  MoveL 3948 to (-81.04, 7.67, -135.54) mm, rotated rx 42.04 ry 15.1 rz -114.75 deg; joints [-14.521, -47.036, 111.718, 147.61, 50.435, -29.895, -355]
  MoveL 3949 to (-78.95, 8.33, -135.66) mm, rotated rx 42.04 ry 15.1 rz -114.75 deg; joints [-14.521, -46.888, 111.628, 147.636, 50.484, -29.936, -355]
  MoveL 3950 to (-78.47, 8.53, -135.68) mm, rotated rx 42.04 ry 15.1 rz -114.75 deg; joints [-14.52, -46.852, 111.603, 147.642, 50.493, -29.944, -355]
  MoveL 3951 to (-78.06, 8.74, -135.73) mm, rotated rx 42.04 ry 15.1 rz -114.75 deg; joints [-14.52, -46.82, 111.578, 147.645, 50.499, -29.949, -355]
  MoveL 3952 to (-77.68, 8.96, -135.8) mm, rotated rx 42.04 ry 15.1 rz -114.75 deg; joints [-14.521, -46.79, 111.553, 147.645, 50.503, -29.951, -355]
  MoveL 3953 to (-77.28, 9.16, -135.86) mm, rotated rx 42.04 ry 15.1 rz -114.75 deg; joints [-14.522, -46.759, 111.528, 147.647, 50.509, -29.956, -355]
  MoveL 3954 to (-76.86, 9.36, -135.89) mm, rotated rx 42.04 ry 15.1 rz -114.75 deg; joints [-14.522, -46.727, 111.504, 147.651, 50.515, -29.961, -355]
  MoveL 3955 to (-72.52, 11.13, -135.9) mm, rotated rx 42.04 ry 15.1 rz -114.75 deg; joints [-14.508, -46.408, 111.285, 147.712, 50.597, -30.037, -355]
  MoveL 3956 to (-72.12, 11.31, -135.92) mm, rotated rx 42.04 ry 15.1 rz -114.75 deg; joints [-14.507, -46.377, 111.263, 147.716, 50.603, -30.043, -355]
  MoveL 3957 to (-71.68, 11.49, -135.93) mm, rotated rx 42.04 ry 15.1 rz -114.75 deg; joints [-14.506, -46.345, 111.24, 147.722, 50.611, -30.05, -355]
  MoveL 3958 to (-70.72, 11.88, -135.93) mm, rotated rx 42.04 ry 15.1 rz -114.75 deg; joints [-14.503, -46.274, 111.191, 147.735, 50.629, -30.066, -355]
  MoveL 3959 to (-70.2, 12.11, -135.94) mm, rotated rx 42.04 ry 15.1 rz -114.75 deg; joints [-14.502, -46.235, 111.163, 147.742, 50.638, -30.075, -355]
  MoveL 3960 to (-69.65, 12.36, -135.96) mm, rotated rx 42.04 ry 15.1 rz -114.75 deg; joints [-14.5, -46.194, 111.132, 147.748, 50.646, -30.082, -355]
  MoveL 3961 to (-69.07, 12.68, -135.99) mm, rotated rx 42.04 ry 15.1 rz -114.75 deg; joints [-14.499, -46.148, 111.095, 147.753, 50.653, -30.089, -355]
  MoveL 3962 to (-68.53, 13.06, -136.01) mm, rotated rx 42.04 ry 15.1 rz -114.75 deg; joints [-14.497, -46.103, 111.053, 147.757, 50.656, -30.092, -355]
  MoveL 3963 to (-68.02, 13.48, -136.03) mm, rotated rx 42.04 ry 15.1 rz -114.75 deg; joints [-14.494, -46.059, 111.009, 147.76, 50.655, -30.093, -355]
  MoveL 3964 to (-69.19, 12.88, -137.01) mm, rotated rx 42.04 ry 15.1 rz -114.75 deg; joints [-14.538, -46.143, 111.064, 147.695, 50.641, -30.053, -355]
  MoveL 3965 to (-68.73, 14.14, -137.43) mm, rotated rx 42.04 ry 15.1 rz -114.75 deg; joints [-14.546, -46.072, 110.943, 147.663, 50.6, -30.014, -355]
  MoveL 3966 to (-68.09, 15.49, -137.75) mm, rotated rx 42.04 ry 15.1 rz -114.75 deg; joints [-14.549, -45.989, 110.812, 147.639, 50.561, -29.981, -355]
  MoveL 3967 to (-67.25, 16.96, -137.99) mm, rotated rx 42.04 ry 15.1 rz -114.75 deg; joints [-14.548, -45.89, 110.669, 147.621, 50.523, -29.95, -355]
  MoveL 3968 to (-66.1, 18.76, -138.21) mm, rotated rx 42.04 ry 15.1 rz -114.75 deg; joints [-14.543, -45.761, 110.493, 147.605, 50.481, -29.919, -355]
  MoveL 3969 to (-64.92, 20.54, -138.32) mm, rotated rx 42.04 ry 15.1 rz -114.75 deg; joints [-14.535, -45.633, 110.319, 147.595, 50.441, -29.892, -355]
  MoveL 3970 to (-63.74, 22.32, -138.43) mm, rotated rx 42.04 ry 15.1 rz -114.75 deg; joints [-14.526, -45.504, 110.145, 147.585, 50.401, -29.864, -355]
  MoveL 3971 to (-62.57, 24.1, -138.66) mm, rotated rx 42.04 ry 15.1 rz -114.75 deg; joints [-14.522, -45.375, 109.968, 147.569, 50.36, -29.833, -355]
  MoveL 3972 to (-61.39, 25.88, -138.78) mm, rotated rx 42.04 ry 15.1 rz -114.75 deg; joints [-14.514, -45.247, 109.794, 147.558, 50.319, -29.805, -355]
  MoveL 3973 to (-60.21, 27.66, -139.01) mm, rotated rx 42.04 ry 15.1 rz -114.75 deg; joints [-14.51, -45.117, 109.617, 147.542, 50.278, -29.773, -355]
  MoveL 3974 to (-59.02, 29.43, -139.12) mm, rotated rx 42.04 ry 15.1 rz -114.75 deg; joints [-14.502, -44.988, 109.442, 147.531, 50.238, -29.745, -355]
  MoveL 3975 to (-57.83, 31.2, -139.24) mm, rotated rx 42.04 ry 15.1 rz -114.75 deg; joints [-14.494, -44.859, 109.267, 147.52, 50.197, -29.717, -355]
  MoveL 3976 to (-56.64, 32.97, -139.48) mm, rotated rx 42.04 ry 15.1 rz -114.75 deg; joints [-14.491, -44.729, 109.09, 147.503, 50.156, -29.686, -355]
  MoveL 3977 to (-55.48, 34.65, -139.58) mm, rotated rx 42.04 ry 15.1 rz -114.75 deg; joints [-14.483, -44.606, 108.923, 147.493, 50.118, -29.659, -355]
  MoveL 3978 to (-54.36, 36.29, -139.79) mm, rotated rx 42.04 ry 15.1 rz -114.75 deg; joints [-14.479, -44.484, 108.758, 147.478, 50.081, -29.63, -355]
  MoveL 3979 to (-53.04, 38.26, -139.95) mm, rotated rx 42.04 ry 15.1 rz -114.75 deg; joints [-14.471, -44.341, 108.562, 147.464, 50.034, -29.597, -355]
  MoveL 3980 to (-51.48, 40.49, -140.04) mm, rotated rx 42.04 ry 15.1 rz -114.75 deg; joints [-14.459, -44.175, 108.339, 147.453, 49.983, -29.563, -355]
  MoveL 3981 to (-50.32, 42.21, -140.1) mm, rotated rx 42.04 ry 15.1 rz -114.75 deg; joints [-14.449, -44.05, 108.168, 147.444, 49.942, -29.535, -355]
  MoveL 3982 to (-49.24, 43.8, -140.23) mm, rotated rx 42.04 ry 15.1 rz -114.75 deg; joints [-14.443, -43.933, 108.008, 147.432, 49.904, -29.508, -355]
  MoveL 3983 to (-48.12, 45.44, -140.34) mm, rotated rx 42.04 ry 15.1 rz -114.75 deg; joints [-14.435, -43.813, 107.844, 147.421, 49.866, -29.481, -355]
  MoveL 3984 to (-47.01, 47.05, -140.45) mm, rotated rx 42.04 ry 15.1 rz -114.75 deg; joints [-14.428, -43.694, 107.682, 147.41, 49.827, -29.453, -355]
  MoveL 3985 to (-45.85, 48.75, -140.52) mm, rotated rx 42.04 ry 15.1 rz -114.75 deg; joints [-14.419, -43.57, 107.511, 147.4, 49.787, -29.426, -355]
  MoveL 3986 to (-44.59, 50.58, -140.62) mm, rotated rx 42.04 ry 15.1 rz -114.75 deg; joints [-14.41, -43.435, 107.327, 147.389, 49.743, -29.395, -355]
  MoveL 3987 to (-43.19, 52.55, -140.88) mm, rotated rx 42.04 ry 15.1 rz -114.75 deg; joints [-14.406, -43.286, 107.125, 147.369, 49.697, -29.359, -355]
  MoveL 3988 to (-42.36, 54.62, -141.86) mm, rotated rx 42.04 ry 15.1 rz -114.75 deg; joints [-14.43, -43.163, 106.913, 147.299, 49.627, -29.284, -355]
  MoveL 3989 to (-42.38, 53.48, -142.35) mm, rotated rx 42.04 ry 15.1 rz -114.75 deg; joints [-14.457, -43.198, 107.005, 147.294, 49.682, -29.312, -355]
  MoveL 3990 to (-42.39, 52.89, -142.66) mm, rotated rx 42.04 ry 15.1 rz -114.75 deg; joints [-14.473, -43.216, 107.053, 147.288, 49.711, -29.326, -355]
  MoveL 3991 to (-42.38, 52.79, -142.81) mm, rotated rx 42.04 ry 15.1 rz -114.75 deg; joints [-14.479, -43.218, 107.059, 147.282, 49.716, -29.325, -355]
  MoveL 3992 to (-42.37, 53.13, -142.85) mm, rotated rx 42.04 ry 15.1 rz -114.75 deg; joints [-14.478, -43.206, 107.028, 147.274, 49.7, -29.312, -355]
  MoveL 3993 to (-42.37, 53.6, -142.86) mm, rotated rx 42.04 ry 15.1 rz -114.75 deg; joints [-14.476, -43.19, 106.987, 147.266, 49.678, -29.296, -355]
  MoveL 3994 to (-42.34, 54.08, -142.9) mm, rotated rx 42.04 ry 15.1 rz -114.75 deg; joints [-14.474, -43.173, 106.944, 147.256, 49.656, -29.278, -355]
  MoveL 3995 to (-42.31, 54.53, -142.96) mm, rotated rx 42.04 ry 15.1 rz -114.75 deg; joints [-14.473, -43.156, 106.903, 147.246, 49.635, -29.262, -355]
  MoveL 3996 to (-42.28, 54.99, -143) mm, rotated rx 42.04 ry 15.1 rz -114.75 deg; joints [-14.471, -43.139, 106.861, 147.237, 49.614, -29.245, -355]
  MoveL 3997 to (-42.26, 55.48, -143.02) mm, rotated rx 42.04 ry 15.1 rz -114.75 deg; joints [-14.469, -43.122, 106.818, 147.228, 49.591, -29.227, -355]
  MoveL 3998 to (-42.25, 58.1, -143.02) mm, rotated rx 42.04 ry 15.1 rz -114.75 deg; joints [-14.451, -43.036, 106.587, 147.182, 49.466, -29.133, -355]
  MoveL 3999 to (-42.24, 58.56, -143.04) mm, rotated rx 42.04 ry 15.1 rz -114.75 deg; joints [-14.449, -43.02, 106.546, 147.174, 49.445, -29.117, -355]
  MoveL 4000 to (-42.21, 58.94, -143.07) mm, rotated rx 42.04 ry 15.1 rz -114.75 deg; joints [-14.448, -43.005, 106.511, 147.166, 49.427, -29.103, -355]
  MoveL 4001 to (-42.19, 59.4, -143.09) mm, rotated rx 42.04 ry 15.1 rz -114.75 deg; joints [-14.445, -42.989, 106.47, 147.157, 49.405, -29.086, -355]
  MoveL 4002 to (-42.18, 60, -143.11) mm, rotated rx 42.04 ry 15.1 rz -114.75 deg; joints [-14.442, -42.968, 106.417, 147.146, 49.377, -29.064, -355]
  MoveL 4003 to (-42.13, 60.72, -143.17) mm, rotated rx 42.04 ry 15.1 rz -114.75 deg; joints [-14.439, -42.942, 106.352, 147.131, 49.344, -29.038, -355]
  MoveL 4004 to (-42.11, 61.34, -143.2) mm, rotated rx 42.04 ry 15.1 rz -114.75 deg; joints [-14.436, -42.92, 106.296, 147.119, 49.315, -29.016, -355]
  MoveL 4005 to (-42.11, 61.87, -143.2) mm, rotated rx 42.04 ry 15.1 rz -114.75 deg; joints [-14.433, -42.902, 106.249, 147.11, 49.29, -28.996, -355]
  MoveL 4006 to (-42.1, 63.44, -143.2) mm, rotated rx 42.04 ry 15.1 rz -114.75 deg; joints [-14.422, -42.849, 106.11, 147.082, 49.215, -28.939, -355]
  MoveL 4007 to (-41.79, 66.34, -143.54) mm, rotated rx 42.04 ry 15.1 rz -114.75 deg; joints [-14.416, -42.733, 105.843, 147.019, 49.086, -28.834, -355]
  MoveL 4008 to (-41.42, 67.58, -143.97) mm, rotated rx 42.04 ry 15.1 rz -114.75 deg; joints [-14.424, -42.667, 105.719, 146.982, 49.04, -28.788, -355]
  MoveL 4009 to (-40.9, 68.68, -144.57) mm, rotated rx 42.04 ry 15.1 rz -114.75 deg; joints [-14.439, -42.596, 105.603, 146.941, 49.006, -28.748, -355]
  MoveL 4010 to (-39.42, 70.47, -146.28) mm, rotated rx 42.04 ry 15.1 rz -114.75 deg; joints [-14.492, -42.439, 105.39, 146.851, 48.972, -28.681, -355]
  MoveL 4011 to (-37.35, 71.7, -148.68) mm, rotated rx 42.04 ry 15.1 rz -114.75 deg; joints [-14.574, -42.261, 105.204, 146.746, 48.986, -28.633, -355]
  MoveL 4012 to (-35.34, 72.15, -151.07) mm, rotated rx 42.04 ry 15.1 rz -114.75 deg; joints [-14.661, -42.113, 105.088, 146.655, 49.035, -28.613, -355]
  MoveL 4013 to (-34.6, 71.99, -152.01) mm, rotated rx 42.04 ry 15.1 rz -114.75 deg; joints [-14.698, -42.068, 105.073, 146.625, 49.069, -28.617, -355]
  MoveL 4014 to (-34.02, 71.57, -152.78) mm, rotated rx 42.04 ry 15.1 rz -114.75 deg; joints [-14.73, -42.044, 105.087, 146.604, 49.109, -28.629, -355]
  MoveL 4015 to (-33.8, 71.26, -153.1) mm, rotated rx 42.04 ry 15.1 rz -114.75 deg; joints [-14.744, -42.039, 105.105, 146.598, 49.132, -28.638, -355]
  MoveL 4016 to (-33.63, 70.89, -153.38) mm, rotated rx 42.04 ry 15.1 rz -114.75 deg; joints [-14.757, -42.039, 105.13, 146.594, 49.156, -28.65, -355]
  MoveL 4017 to (-33.4, 69.96, -153.81) mm, rotated rx 42.04 ry 15.1 rz -114.75 deg; joints [-14.78, -42.054, 105.202, 146.593, 49.209, -28.68, -355]
  MoveL 4018 to (-33.35, 68.77, -154.07) mm, rotated rx 42.04 ry 15.1 rz -114.75 deg; joints [-14.798, -42.088, 105.302, 146.603, 49.268, -28.719, -355]
  MoveL 4019 to (-33.47, 67.32, -154.15) mm, rotated rx 42.04 ry 15.1 rz -114.75 deg; joints [-14.811, -42.143, 105.431, 146.622, 49.334, -28.767, -355]
  MoveL 4020 to (-33.54, 66.8, -154.15) mm, rotated rx 42.04 ry 15.1 rz -114.75 deg; joints [-14.815, -42.164, 105.479, 146.63, 49.357, -28.784, -355]
  MoveL 4021 to (-33.64, 66.37, -154.1) mm, rotated rx 42.04 ry 15.1 rz -114.75 deg; joints [-14.816, -42.184, 105.519, 146.639, 49.374, -28.798, -355]
  MoveL 4022 to (-33.74, 65.95, -154.04) mm, rotated rx 42.04 ry 15.1 rz -114.75 deg; joints [-14.816, -42.204, 105.56, 146.647, 49.391, -28.813, -355]
  MoveL 4023 to (-33.82, 65.49, -154) mm, rotated rx 42.04 ry 15.1 rz -114.75 deg; joints [-14.818, -42.225, 105.603, 146.656, 49.41, -28.828, -355]
  MoveL 4024 to (-33.9, 65, -153.98) mm, rotated rx 42.04 ry 15.1 rz -114.75 deg; joints [-14.821, -42.246, 105.648, 146.664, 49.431, -28.844, -355]
  MoveL 4025 to (-33.98, 64.47, -153.98) mm, rotated rx 42.04 ry 15.1 rz -114.75 deg; joints [-14.824, -42.267, 105.697, 146.672, 49.454, -28.862, -355]
  MoveL 4026 to (-34.05, 63.95, -153.98) mm, rotated rx 42.04 ry 15.1 rz -114.75 deg; joints [-14.828, -42.288, 105.744, 146.68, 49.477, -28.879, -355]
  MoveL 4027 to (-34.1, 63.44, -153.99) mm, rotated rx 42.04 ry 15.1 rz -114.75 deg; joints [-14.832, -42.308, 105.789, 146.687, 49.5, -28.895, -355]
  MoveL 4028 to (-34.16, 62.95, -154) mm, rotated rx 42.04 ry 15.1 rz -114.75 deg; joints [-14.836, -42.327, 105.834, 146.694, 49.522, -28.912, -355]
  MoveL 4029 to (-34.23, 62.49, -153.98) mm, rotated rx 42.04 ry 15.1 rz -114.75 deg; joints [-14.838, -42.347, 105.876, 146.702, 49.541, -28.927, -355]
  MoveL 4030 to (-34.31, 62.04, -153.94) mm, rotated rx 42.04 ry 15.1 rz -114.75 deg; joints [-14.84, -42.367, 105.918, 146.71, 49.56, -28.942, -355]
  MoveL 4031 to (-34.42, 61.5, -153.89) mm, rotated rx 42.04 ry 15.1 rz -114.75 deg; joints [-14.842, -42.391, 105.968, 146.72, 49.582, -28.96, -355]
  MoveL 4032 to (-34.55, 60.81, -153.84) mm, rotated rx 42.04 ry 15.1 rz -114.75 deg; joints [-14.845, -42.422, 106.033, 146.732, 49.611, -28.983, -355]
  MoveL 4033 to (-34.66, 60.18, -153.81) mm, rotated rx 42.04 ry 15.1 rz -114.75 deg; joints [-14.848, -42.449, 106.091, 146.743, 49.638, -29.003, -355]
  MoveL 4034 to (-35.01, 57.58, -153.81) mm, rotated rx 42.04 ry 15.1 rz -114.75 deg; joints [-14.867, -42.554, 106.326, 146.781, 49.751, -29.088, -355]
  MoveL 4035 to (-35.11, 56.96, -153.78) mm, rotated rx 42.04 ry 15.1 rz -114.75 deg; joints [-14.869, -42.58, 106.383, 146.792, 49.777, -29.109, -355]
  MoveL 4036 to (-35.21, 56.41, -153.72) mm, rotated rx 42.04 ry 15.1 rz -114.75 deg; joints [-14.871, -42.604, 106.434, 146.802, 49.801, -29.127, -355]
  MoveL 4037 to (-35.25, 56.21, -153.57) mm, rotated rx 42.04 ry 15.1 rz -114.75 deg; joints [-14.867, -42.615, 106.455, 146.812, 49.809, -29.137, -355]
  MoveL 4038 to (-35.23, 56.33, -153.31) mm, rotated rx 42.04 ry 15.1 rz -114.75 deg; joints [-14.856, -42.611, 106.448, 146.824, 49.803, -29.14, -355]
  MoveL 4039 to (-35.13, 56.78, -152.9) mm, rotated rx 42.04 ry 15.1 rz -114.75 deg; joints [-14.837, -42.594, 106.414, 146.839, 49.784, -29.137, -355]
  MoveL 4040 to (-36.15, 56.59, -152.1) mm, rotated rx 42.04 ry 15.1 rz -114.75 deg; joints [-14.808, -42.665, 106.463, 146.863, 49.759, -29.135, -355]
  MoveL 4041 to (-37.5, 55.14, -151.88) mm, rotated rx 42.04 ry 15.1 rz -114.75 deg; joints [-14.81, -42.794, 106.619, 146.873, 49.782, -29.153, -355]
  MoveL 4042 to (-38.85, 53.66, -151.72) mm, rotated rx 42.04 ry 15.1 rz -114.75 deg; joints [-14.815, -42.923, 106.776, 146.881, 49.807, -29.171, -355]
  MoveL 4043 to (-40.23, 52.13, -151.57) mm, rotated rx 42.04 ry 15.1 rz -114.75 deg; joints [-14.821, -43.055, 106.938, 146.888, 49.833, -29.19, -355]
  MoveL 4044 to (-41.5, 50.75, -151.28) mm, rotated rx 42.04 ry 15.1 rz -114.75 deg; joints [-14.82, -43.177, 107.087, 146.902, 49.856, -29.21, -355]
  MoveL 4045 to (-42.91, 49.19, -151.09) mm, rotated rx 42.04 ry 15.1 rz -114.75 deg; joints [-14.824, -43.313, 107.253, 146.91, 49.882, -29.229, -355]
  MoveL 4046 to (-44.4, 47.54, -150.9) mm, rotated rx 42.04 ry 15.1 rz -114.75 deg; joints [-14.829, -43.456, 107.427, 146.918, 49.909, -29.249, -355]
  MoveL 4047 to (-45.9, 45.87, -150.82) mm, rotated rx 42.04 ry 15.1 rz -114.75 deg; joints [-14.838, -43.599, 107.601, 146.922, 49.937, -29.266, -355]
  MoveL 4048 to (-47.71, 43.83, -150.73) mm, rotated rx 42.04 ry 15.1 rz -114.75 deg; joints [-14.85, -43.774, 107.813, 146.925, 49.971, -29.288, -355]
  MoveL 4049 to (-49.01, 42.36, -150.62) mm, rotated rx 42.04 ry 15.1 rz -114.75 deg; joints [-14.857, -43.899, 107.966, 146.929, 49.996, -29.304, -355]
  MoveL 4050 to (-50.22, 41, -150.41) mm, rotated rx 42.04 ry 15.1 rz -114.75 deg; joints [-14.859, -44.017, 108.11, 146.939, 50.018, -29.322, -355]
  MoveL 4051 to (-51.55, 39.48, -150.22) mm, rotated rx 42.04 ry 15.1 rz -114.75 deg; joints [-14.862, -44.146, 108.268, 146.947, 50.043, -29.34, -355]
  MoveL 4052 to (-52.96, 37.88, -150.1) mm, rotated rx 42.04 ry 15.1 rz -114.75 deg; joints [-14.87, -44.283, 108.434, 146.951, 50.069, -29.357, -355]
  MoveL 4053 to (-54.35, 36.29, -149.92) mm, rotated rx 42.04 ry 15.1 rz -114.75 deg; joints [-14.875, -44.419, 108.599, 146.959, 50.095, -29.376, -355]
  MoveL 4054 to (-55.74, 34.7, -149.8) mm, rotated rx 42.04 ry 15.1 rz -114.75 deg; joints [-14.882, -44.554, 108.763, 146.963, 50.121, -29.393, -355]
  MoveL 4055 to (-57.17, 33.05, -149.62) mm, rotated rx 42.04 ry 15.1 rz -114.75 deg; joints [-14.887, -44.693, 108.933, 146.97, 50.148, -29.412, -355]
  MoveL 4056 to (-58.57, 31.44, -149.5) mm, rotated rx 42.04 ry 15.1 rz -114.75 deg; joints [-14.895, -44.83, 109.098, 146.974, 50.174, -29.429, -355]
  MoveL 4057 to (-59.96, 29.82, -149.27) mm, rotated rx 42.04 ry 15.1 rz -114.75 deg; joints [-14.898, -44.966, 109.265, 146.985, 50.2, -29.449, -355]
  MoveL 4058 to (-61.36, 28.2, -149.16) mm, rotated rx 42.04 ry 15.1 rz -114.75 deg; joints [-14.906, -45.103, 109.43, 146.988, 50.226, -29.465, -355]
  MoveL 4059 to (-62.75, 26.59, -149.04) mm, rotated rx 42.04 ry 15.1 rz -114.75 deg; joints [-14.914, -45.239, 109.595, 146.992, 50.251, -29.482, -355]
  MoveL 4060 to (-64.13, 24.95, -148.82) mm, rotated rx 42.04 ry 15.1 rz -114.75 deg; joints [-14.917, -45.376, 109.762, 147.001, 50.278, -29.502, -355]
  MoveL 4061 to (-65.34, 23.44, -148.61) mm, rotated rx 42.04 ry 15.1 rz -114.75 deg; joints [-14.921, -45.498, 109.915, 147.011, 50.305, -29.522, -355]
  MoveL 4062 to (-66.39, 22.03, -148.32) mm, rotated rx 42.04 ry 15.1 rz -114.75 deg; joints [-14.92, -45.609, 110.059, 147.027, 50.332, -29.546, -355]
  MoveL 4063 to (-67.29, 20.67, -147.92) mm, rotated rx 42.04 ry 15.1 rz -114.75 deg; joints [-14.914, -45.71, 110.197, 147.05, 50.362, -29.575, -355]
  MoveL 4064 to (-65.98, 21.37, -146.99) mm, rotated rx 42.04 ry 15.1 rz -114.75 deg; joints [-14.872, -45.614, 110.13, 147.114, 50.376, -29.614, -355]
  MoveL 4065 to (-66.44, 21.02, -146.98) mm, rotated rx 42.04 ry 15.1 rz -114.75 deg; joints [-14.874, -45.653, 110.167, 147.11, 50.375, -29.612, -355]
  MoveL 4066 to (-66.89, 20.74, -146.96) mm, rotated rx 42.04 ry 15.1 rz -114.75 deg; joints [-14.876, -45.69, 110.2, 147.107, 50.372, -29.609, -355]
  MoveL 4067 to (-67.31, 20.52, -146.9) mm, rotated rx 42.04 ry 15.1 rz -114.75 deg; joints [-14.875, -45.722, 110.226, 147.105, 50.367, -29.605, -355]
  MoveL 4068 to (-67.71, 20.33, -146.83) mm, rotated rx 42.04 ry 15.1 rz -114.75 deg; joints [-14.874, -45.753, 110.25, 147.103, 50.361, -29.601, -355]
  MoveL 4069 to (-68.15, 20.17, -146.78) mm, rotated rx 42.04 ry 15.1 rz -114.75 deg; joints [-14.873, -45.785, 110.272, 147.099, 50.352, -29.594, -355]
  MoveL 4070 to (-68.61, 20.02, -146.75) mm, rotated rx 42.04 ry 15.1 rz -114.75 deg; joints [-14.873, -45.818, 110.293, 147.094, 50.342, -29.585, -355]
  MoveL 4071 to (-69.12, 19.87, -146.73) mm, rotated rx 42.04 ry 15.1 rz -114.75 deg; joints [-14.874, -45.853, 110.314, 147.087, 50.33, -29.575, -355]
  MoveL 4072 to (-69.63, 19.74, -146.73) mm, rotated rx 42.04 ry 15.1 rz -114.75 deg; joints [-14.875, -45.887, 110.333, 147.079, 50.318, -29.564, -355]
  MoveL 4073 to (-70.08, 19.61, -146.72) mm, rotated rx 42.04 ry 15.1 rz -114.75 deg; joints [-14.876, -45.919, 110.352, 147.072, 50.308, -29.554, -355]
  MoveL 4074 to (-70.48, 19.48, -146.69) mm, rotated rx 42.04 ry 15.1 rz -114.75 deg; joints [-14.876, -45.947, 110.37, 147.067, 50.299, -29.547, -355]
  MoveL 4075 to (-70.94, 19.34, -146.68) mm, rotated rx 42.04 ry 15.1 rz -114.75 deg; joints [-14.877, -45.98, 110.389, 147.06, 50.288, -29.537, -355]
  MoveL 4076 to (-71.45, 19.21, -146.68) mm, rotated rx 42.04 ry 15.1 rz -114.75 deg; joints [-14.878, -46.014, 110.409, 147.052, 50.276, -29.526, -355]
  MoveL 4077 to (-72.04, 19.04, -146.66) mm, rotated rx 42.04 ry 15.1 rz -114.75 deg; joints [-14.879, -46.055, 110.433, 147.044, 50.262, -29.514, -355]
  MoveL 4078 to (-72.7, 18.85, -146.62) mm, rotated rx 42.04 ry 15.1 rz -114.75 deg; joints [-14.879, -46.102, 110.461, 147.035, 50.246, -29.501, -355]
  MoveL 4079 to (-73.29, 18.68, -146.6) mm, rotated rx 42.04 ry 15.1 rz -114.75 deg; joints [-14.879, -46.143, 110.485, 147.027, 50.232, -29.489, -355]
  MoveL 4080 to (-73.9, 18.5, -146.57) mm, rotated rx 42.04 ry 15.1 rz -114.75 deg; joints [-14.88, -46.186, 110.511, 147.018, 50.218, -29.476, -355]
  MoveL 4081 to (-74.58, 18.29, -146.53) mm, rotated rx 42.04 ry 15.1 rz -114.75 deg; joints [-14.88, -46.234, 110.541, 147.01, 50.203, -29.463, -355]
  MoveL 4082 to (-75.15, 18.12, -146.52) mm, rotated rx 42.04 ry 15.1 rz -114.75 deg; joints [-14.881, -46.273, 110.564, 147.001, 50.189, -29.451, -355]
  MoveL 4083 to (-75.68, 17.98, -146.52) mm, rotated rx 42.04 ry 15.1 rz -114.75 deg; joints [-14.882, -46.309, 110.584, 146.993, 50.176, -29.439, -355]
  MoveL 4084 to (-77.2, 17.58, -146.52) mm, rotated rx 42.04 ry 15.1 rz -114.75 deg; joints [-14.886, -46.414, 110.642, 146.967, 50.138, -29.405, -355]
  MoveL 4085 to (-78.62, 17.28, -146.6) mm, rotated rx 42.04 ry 15.1 rz -114.75 deg; joints [-14.892, -46.508, 110.689, 146.938, 50.1, -29.368, -355]
  MoveL 4086 to (-79.8, 17.18, -146.85) mm, rotated rx 42.04 ry 15.1 rz -114.75 deg; joints [-14.903, -46.581, 110.711, 146.902, 50.06, -29.327, -355]
  MoveL 4087 to (-80.75, 17.29, -147.28) mm, rotated rx 42.04 ry 15.1 rz -114.75 deg; joints [-14.92, -46.632, 110.71, 146.858, 50.021, -29.282, -355]
  MoveL 4088 to (-81.14, 17.42, -147.55) mm, rotated rx 42.04 ry 15.1 rz -114.75 deg; joints [-14.93, -46.649, 110.701, 146.834, 50.001, -29.258, -355]
  MoveL 4089 to (-81.47, 17.6, -147.87) mm, rotated rx 42.04 ry 15.1 rz -114.75 deg; joints [-14.941, -46.661, 110.685, 146.807, 49.981, -29.233, -355]
  MoveL 4090 to (-81.96, 18.11, -148.63) mm, rotated rx 42.04 ry 15.1 rz -114.75 deg; joints [-14.968, -46.668, 110.637, 146.75, 49.94, -29.18, -355]
  MoveL 4091 to (-82.21, 18.83, -149.55) mm, rotated rx 42.04 ry 15.1 rz -114.75 deg; joints [-14.999, -46.653, 110.564, 146.685, 49.9, -29.124, -355]
  MoveL 4092 to (-82.01, 20.88, -151.92) mm, rotated rx 42.04 ry 15.1 rz -114.75 deg; joints [-15.078, -46.558, 110.347, 146.534, 49.817, -28.998, -355]
  MoveL 4093 to (-81.03, 23.07, -154.28) mm, rotated rx 42.04 ry 15.1 rz -114.75 deg; joints [-15.154, -46.412, 110.105, 146.397, 49.756, -28.892, -355]
  MoveL 4094 to (-79.44, 24.76, -155.97) mm, rotated rx 42.04 ry 15.1 rz -114.75 deg; joints [-15.207, -46.249, 109.908, 146.316, 49.74, -28.841, -355]
  MoveL 4095 to (-78.41, 25.41, -156.56) mm, rotated rx 42.04 ry 15.1 rz -114.75 deg; joints [-15.225, -46.162, 109.826, 146.297, 49.749, -28.836, -355]
  MoveL 4096 to (-77.22, 25.94, -156.98) mm, rotated rx 42.04 ry 15.1 rz -114.75 deg; joints [-15.237, -46.071, 109.756, 146.292, 49.769, -28.845, -355]
  MoveL 4097 to (-74.38, 26.6, -157.32) mm, rotated rx 42.04 ry 15.1 rz -114.75 deg; joints [-15.244, -45.878, 109.649, 146.324, 49.842, -28.905, -355]
  MoveL 4098 to (-70.23, 27.14, -157.32) mm, rotated rx 42.04 ry 15.1 rz -114.75 deg; joints [-15.238, -45.613, 109.536, 146.402, 49.968, -29.018, -355]
  MoveL 4099 to (-69.68, 27.22, -157.34) mm, rotated rx 42.04 ry 15.1 rz -114.75 deg; joints [-15.238, -45.577, 109.52, 146.411, 49.983, -29.032, -355]
  MoveL 4100 to (-69.16, 27.32, -157.37) mm, rotated rx 42.04 ry 15.1 rz -114.75 deg; joints [-15.239, -45.543, 109.502, 146.418, 49.998, -29.044, -355]
  MoveL 4101 to (-68.64, 27.43, -157.44) mm, rotated rx 42.04 ry 15.1 rz -114.75 deg; joints [-15.24, -45.508, 109.483, 146.424, 50.011, -29.055, -355]
  MoveL 4102 to (-68.14, 27.55, -157.52) mm, rotated rx 42.04 ry 15.1 rz -114.75 deg; joints [-15.242, -45.473, 109.463, 146.428, 50.024, -29.064, -355]
  MoveL 4103 to (-67.65, 27.67, -157.6) mm, rotated rx 42.04 ry 15.1 rz -114.75 deg; joints [-15.244, -45.439, 109.443, 146.433, 50.036, -29.074, -355]
  MoveL 4104 to (-67.17, 27.76, -157.64) mm, rotated rx 42.04 ry 15.1 rz -114.75 deg; joints [-15.245, -45.408, 109.427, 146.439, 50.049, -29.084, -355]
  MoveL 4105 to (-66.7, 27.83, -157.65) mm, rotated rx 42.04 ry 15.1 rz -114.75 deg; joints [-15.245, -45.377, 109.413, 146.447, 50.063, -29.096, -355]
  MoveL 4106 to (-66.18, 27.9, -157.65) mm, rotated rx 42.04 ry 15.1 rz -114.75 deg; joints [-15.244, -45.344, 109.399, 146.457, 50.079, -29.11, -355]
  MoveL 4107 to (-65.56, 28, -157.69) mm, rotated rx 42.04 ry 15.1 rz -114.75 deg; joints [-15.244, -45.303, 109.379, 146.466, 50.096, -29.125, -355]
  MoveL 4108 to (-64.89, 28.13, -157.75) mm, rotated rx 42.04 ry 15.1 rz -114.75 deg; joints [-15.245, -45.259, 109.356, 146.475, 50.115, -29.141, -355]
  MoveL 4109 to (-64.3, 28.24, -157.77) mm, rotated rx 42.04 ry 15.1 rz -114.75 deg; joints [-15.245, -45.22, 109.336, 146.484, 50.13, -29.154, -355]
  MoveL 4110 to (-63.77, 28.39, -157.78) mm, rotated rx 42.04 ry 15.1 rz -114.75 deg; joints [-15.244, -45.183, 109.315, 146.492, 50.143, -29.166, -355]
  MoveL 4111 to (-63.25, 28.58, -157.78) mm, rotated rx 42.04 ry 15.1 rz -114.75 deg; joints [-15.242, -45.146, 109.289, 146.499, 50.152, -29.175, -355]
  MoveL 4112 to (-62.76, 28.89, -157.78) mm, rotated rx 42.04 ry 15.1 rz -114.75 deg; joints [-15.24, -45.107, 109.255, 146.504, 50.155, -29.179, -355]
  MoveL 4113 to (-62.28, 29.27, -157.78) mm, rotated rx 42.04 ry 15.1 rz -114.75 deg; joints [-15.237, -45.066, 109.214, 146.508, 50.154, -29.181, -355]
  MoveL 4114 to (-63.7, 28.59, -158.74) mm, rotated rx 42.04 ry 15.1 rz -114.75 deg; joints [-15.28, -45.166, 109.281, 146.441, 50.137, -29.136, -355]
  MoveL 4115 to (-62.93, 29.57, -159.16) mm, rotated rx 42.04 ry 15.1 rz -114.75 deg; joints [-15.289, -45.086, 109.176, 146.419, 50.119, -29.115, -355]
  MoveL 4116 to (-61.98, 30.62, -159.49) mm, rotated rx 42.04 ry 15.1 rz -114.75 deg; joints [-15.293, -44.993, 109.064, 146.405, 50.105, -29.099, -355]
  MoveL 4117 to (-60.84, 31.75, -159.74) mm, rotated rx 42.04 ry 15.1 rz -114.75 deg; joints [-15.294, -44.886, 108.943, 146.397, 50.093, -29.088, -355]
  MoveL 4118 to (-59.25, 33.17, -159.85) mm, rotated rx 42.04 ry 15.1 rz -114.75 deg; joints [-15.287, -44.745, 108.791, 146.401, 50.082, -29.084, -355]
  MoveL 4119 to (-57.68, 34.61, -160.08) mm, rotated rx 42.04 ry 15.1 rz -114.75 deg; joints [-15.285, -44.603, 108.636, 146.398, 50.071, -29.076, -355]
  MoveL 4120 to (-56.09, 36.03, -160.19) mm, rotated rx 42.04 ry 15.1 rz -114.75 deg; joints [-15.278, -44.461, 108.484, 146.401, 50.06, -29.071, -355]
  MoveL 4121 to (-54.49, 37.45, -160.31) mm, rotated rx 42.04 ry 15.1 rz -114.75 deg; joints [-15.271, -44.319, 108.331, 146.404, 50.05, -29.066, -355]
  MoveL 4122 to (-52.91, 38.87, -160.54) mm, rotated rx 42.04 ry 15.1 rz -114.75 deg; joints [-15.269, -44.177, 108.176, 146.4, 50.038, -29.058, -355]
  MoveL 4123 to (-51.31, 40.28, -160.66) mm, rotated rx 42.04 ry 15.1 rz -114.75 deg; joints [-15.262, -44.036, 108.023, 146.403, 50.027, -29.053, -355]
  MoveL 4124 to (-49.71, 41.7, -160.78) mm, rotated rx 42.04 ry 15.1 rz -114.75 deg; joints [-15.256, -43.894, 107.87, 146.405, 50.016, -29.048, -355]
  MoveL 4125 to (-47.87, 43.33, -160.94) mm, rotated rx 42.04 ry 15.1 rz -114.75 deg; joints [-15.249, -43.731, 107.693, 146.407, 50.003, -29.041, -355]
  MoveL 4126 to (-46.29, 44.71, -161.14) mm, rotated rx 42.04 ry 15.1 rz -114.75 deg; joints [-15.246, -43.591, 107.541, 146.405, 49.992, -29.034, -355]
  MoveL 4127 to (-44.55, 46.23, -161.33) mm, rotated rx 42.04 ry 15.1 rz -114.75 deg; joints [-15.242, -43.437, 107.373, 146.404, 49.979, -29.026, -355]
  MoveL 4128 to (-42.84, 47.72, -161.59) mm, rotated rx 42.04 ry 15.1 rz -114.75 deg; joints [-15.24, -43.286, 107.208, 146.4, 49.967, -29.017, -355]
  MoveL 4129 to (-41.24, 49.12, -161.71) mm, rotated rx 42.04 ry 15.1 rz -114.75 deg; joints [-15.233, -43.144, 107.054, 146.402, 49.955, -29.011, -355]
  MoveL 4130 to (-39.63, 50.52, -161.71) mm, rotated rx 42.04 ry 15.1 rz -114.75 deg; joints [-15.222, -43.004, 106.902, 146.409, 49.943, -29.007, -355]
  MoveL 4131 to (-38.04, 51.9, -161.78) mm, rotated rx 42.04 ry 15.1 rz -114.75 deg; joints [-15.215, -42.864, 106.75, 146.413, 49.931, -29.002, -355]
  MoveL 4132 to (-36.47, 53.24, -162) mm, rotated rx 42.04 ry 15.1 rz -114.75 deg; joints [-15.212, -42.727, 106.6, 146.41, 49.92, -28.995, -355]
  MoveL 4133 to (-34.71, 54.71, -162.35) mm, rotated rx 42.04 ry 15.1 rz -114.75 deg; joints [-15.214, -42.572, 106.431, 146.401, 49.909, -28.984, -355]
  MoveL 4134 to (-33.32, 55.87, -162.56) mm, rotated rx 42.04 ry 15.1 rz -114.75 deg; joints [-15.213, -42.451, 106.3, 146.398, 49.9, -28.976, -355]
  MoveL 4135 to (-31.42, 57.43, -162.86) mm, rotated rx 42.04 ry 15.1 rz -114.75 deg; joints [-15.213, -42.286, 106.122, 146.392, 49.889, -28.967, -355]
  MoveL 4136 to (-29.74, 58.86, -162.96) mm, rotated rx 42.04 ry 15.1 rz -114.75 deg; joints [-15.205, -42.139, 105.962, 146.395, 49.876, -28.961, -355]
  MoveL 4137 to (-28.14, 60.26, -162.98) mm, rotated rx 42.04 ry 15.1 rz -114.75 deg; joints [-15.195, -41.999, 105.807, 146.4, 49.861, -28.955, -355]
  MoveL 4138 to (-27.25, 60.37, -163.77) mm, rotated rx 42.04 ry 15.1 rz -114.75 deg; joints [-15.224, -41.938, 105.767, 146.375, 49.886, -28.957, -355]
  MoveL 4139 to (-27.44, 59.97, -164.16) mm, rotated rx 42.04 ry 15.1 rz -114.75 deg; joints [-15.242, -41.959, 105.799, 146.359, 49.899, -28.956, -355]
  MoveL 4140 to (-27.51, 59.85, -164.4) mm, rotated rx 42.04 ry 15.1 rz -114.75 deg; joints [-15.252, -41.966, 105.807, 146.347, 49.903, -28.952, -355]
  MoveL 4141 to (-27.47, 59.99, -164.53) mm, rotated rx 42.04 ry 15.1 rz -114.75 deg; joints [-15.256, -41.958, 105.792, 146.339, 49.898, -28.945, -355]
  MoveL 4142 to (-27.36, 60.37, -164.55) mm, rotated rx 42.04 ry 15.1 rz -114.75 deg; joints [-15.254, -41.939, 105.756, 146.334, 49.883, -28.934, -355]
  MoveL 4143 to (-27.23, 60.82, -164.56) mm, rotated rx 42.04 ry 15.1 rz -114.75 deg; joints [-15.251, -41.917, 105.714, 146.328, 49.866, -28.921, -355]
  MoveL 4144 to (-26.82, 62.33, -164.56) mm, rotated rx 42.04 ry 15.1 rz -114.75 deg; joints [-15.24, -41.843, 105.572, 146.309, 49.806, -28.876, -355]
  MoveL 4145 to (-26.67, 62.87, -164.58) mm, rotated rx 42.04 ry 15.1 rz -114.75 deg; joints [-15.237, -41.817, 105.522, 146.302, 49.786, -28.861, -355]
  MoveL 4146 to (-26.49, 63.39, -164.62) mm, rotated rx 42.04 ry 15.1 rz -114.75 deg; joints [-15.235, -41.789, 105.471, 146.294, 49.766, -28.845, -355]
  MoveL 4147 to (-26.29, 63.93, -164.7) mm, rotated rx 42.04 ry 15.1 rz -114.75 deg; joints [-15.234, -41.76, 105.419, 146.284, 49.747, -28.829, -355]
  MoveL 4148 to (-26.11, 64.45, -164.76) mm, rotated rx 42.04 ry 15.1 rz -114.75 deg; joints [-15.232, -41.731, 105.368, 146.275, 49.727, -28.813, -355]
  MoveL 4149 to (-25.96, 64.96, -164.79) mm, rotated rx 42.04 ry 15.1 rz -114.75 deg; joints [-15.23, -41.706, 105.319, 146.268, 49.708, -28.798, -355]
  MoveL 4150 to (-25.82, 65.43, -164.81) mm, rotated rx 42.04 ry 15.1 rz -114.75 deg; joints [-15.227, -41.682, 105.274, 146.261, 49.69, -28.784, -355]
  MoveL 4151 to (-25.67, 65.87, -164.85) mm, rotated rx 42.04 ry 15.1 rz -114.75 deg; joints [-15.225, -41.658, 105.232, 146.254, 49.674, -28.771, -355]
  MoveL 4152 to (-25.53, 66.29, -164.89) mm, rotated rx 42.04 ry 15.1 rz -114.75 deg; joints [-15.224, -41.636, 105.192, 146.247, 49.658, -28.758, -355]
  MoveL 4153 to (-25.39, 66.76, -164.91) mm, rotated rx 42.04 ry 15.1 rz -114.75 deg; joints [-15.221, -41.612, 105.146, 146.241, 49.639, -28.744, -355]
  MoveL 4154 to (-25.22, 67.33, -164.93) mm, rotated rx 42.04 ry 15.1 rz -114.75 deg; joints [-15.217, -41.584, 105.093, 146.233, 49.618, -28.727, -355]
  MoveL 4155 to (-25, 67.99, -164.98) mm, rotated rx 42.04 ry 15.1 rz -114.75 deg; joints [-15.215, -41.549, 105.029, 146.223, 49.593, -28.707, -355]
  MoveL 4156 to (-24.82, 68.57, -165.01) mm, rotated rx 42.04 ry 15.1 rz -114.75 deg; joints [-15.211, -41.519, 104.973, 146.214, 49.571, -28.69, -355]
  MoveL 4157 to (-24.28, 70.6, -165.01) mm, rotated rx 42.04 ry 15.1 rz -114.75 deg; joints [-15.197, -41.421, 104.782, 146.188, 49.49, -28.63, -355]
  MoveL 4158 to (-23.25, 73.33, -165.34) mm, rotated rx 42.04 ry 15.1 rz -114.75 deg; joints [-15.189, -41.269, 104.514, 146.142, 49.392, -28.548, -355]
  MoveL 4159 to (-22.58, 74.43, -165.75) mm, rotated rx 42.04 ry 15.1 rz -114.75 deg; joints [-15.197, -41.19, 104.395, 146.114, 49.36, -28.515, -355]
  MoveL 4160 to (-21.81, 75.37, -166.33) mm, rotated rx 42.04 ry 15.1 rz -114.75 deg; joints [-15.211, -41.11, 104.286, 146.082, 49.34, -28.487, -355]
  MoveL 4161 to (-19.95, 76.73, -167.98) mm, rotated rx 42.04 ry 15.1 rz -114.75 deg; joints [-15.263, -40.944, 104.1, 146.009, 49.336, -28.446, -355]
  MoveL 4162 to (-17.67, 77.41, -170.29) mm, rotated rx 42.04 ry 15.1 rz -114.75 deg; joints [-15.344, -40.772, 103.954, 145.923, 49.378, -28.425, -355]
  MoveL 4163 to (-15.64, 77.34, -172.59) mm, rotated rx 42.04 ry 15.1 rz -114.75 deg; joints [-15.431, -40.64, 103.879, 145.846, 49.447, -28.425, -355]
  MoveL 4164 to (-14.98, 76.99, -173.5) mm, rotated rx 42.04 ry 15.1 rz -114.75 deg; joints [-15.467, -40.606, 103.88, 145.819, 49.486, -28.433, -355]
  MoveL 4165 to (-14.54, 76.45, -174.24) mm, rotated rx 42.04 ry 15.1 rz -114.75 deg; joints [-15.499, -40.593, 103.907, 145.8, 49.527, -28.447, -355]
  MoveL 4166 to (-14.41, 76.1, -174.55) mm, rotated rx 42.04 ry 15.1 rz -114.75 deg; joints [-15.513, -40.594, 103.93, 145.793, 49.548, -28.456, -355]
  MoveL 4167 to (-14.34, 75.69, -174.82) mm, rotated rx 42.04 ry 15.1 rz -114.75 deg; joints [-15.526, -40.601, 103.96, 145.788, 49.57, -28.467, -355]
  MoveL 4168 to (-14.36, 74.74, -175.23) mm, rotated rx 42.04 ry 15.1 rz -114.75 deg; joints [-15.548, -40.631, 104.039, 145.785, 49.616, -28.492, -355]
  MoveL 4169 to (-14.62, 73.58, -175.48) mm, rotated rx 42.04 ry 15.1 rz -114.75 deg; joints [-15.566, -40.682, 104.143, 145.788, 49.665, -28.522, -355]
  MoveL 4170 to (-15.11, 72.21, -175.56) mm, rotated rx 42.04 ry 15.1 rz -114.75 deg; joints [-15.58, -40.755, 104.273, 145.799, 49.716, -28.558, -355]
  MoveL 4171 to (-16.5, 68.82, -175.56) mm, rotated rx 42.04 ry 15.1 rz -114.75 deg; joints [-15.605, -40.947, 104.603, 145.834, 49.836, -28.647, -355]
  MoveL 4172 to (-16.69, 68.4, -175.54) mm, rotated rx 42.04 ry 15.1 rz -114.75 deg; joints [-15.608, -40.972, 104.644, 145.838, 49.85, -28.658, -355]
  MoveL 4173 to (-16.86, 68.02, -175.52) mm, rotated rx 42.04 ry 15.1 rz -114.75 deg; joints [-15.61, -40.995, 104.681, 145.843, 49.863, -28.668, -355]
  MoveL 4174 to (-17.05, 67.59, -175.5) mm, rotated rx 42.04 ry 15.1 rz -114.75 deg; joints [-15.612, -41.02, 104.724, 145.848, 49.878, -28.679, -355]
  MoveL 4175 to (-18.44, 64.2, -175.5) mm, rotated rx 42.04 ry 15.1 rz -114.75 deg; joints [-15.638, -41.212, 105.052, 145.881, 49.997, -28.767, -355]
  MoveL 4176 to (-18.67, 63.71, -175.48) mm, rotated rx 42.04 ry 15.1 rz -114.75 deg; joints [-15.641, -41.241, 105.101, 145.887, 50.013, -28.779, -355]
  MoveL 4177 to (-18.92, 63.23, -175.44) mm, rotated rx 42.04 ry 15.1 rz -114.75 deg; joints [-15.644, -41.272, 105.149, 145.892, 50.029, -28.791, -355]
  MoveL 4178 to (-19.19, 62.82, -175.4) mm, rotated rx 42.04 ry 15.1 rz -114.75 deg; joints [-15.645, -41.302, 105.191, 145.896, 50.04, -28.8, -355]
  MoveL 4179 to (-19.44, 62.52, -175.33) mm, rotated rx 42.04 ry 15.1 rz -114.75 deg; joints [-15.645, -41.326, 105.224, 145.9, 50.046, -28.806, -355]
  MoveL 4180 to (-19.58, 62.39, -175.17) mm, rotated rx 42.04 ry 15.1 rz -114.75 deg; joints [-15.64, -41.34, 105.24, 145.908, 50.047, -28.81, -355]
  MoveL 4181 to (-19.62, 62.4, -174.84) mm, rotated rx 42.04 ry 15.1 rz -114.75 deg; joints [-15.627, -41.344, 105.246, 145.924, 50.046, -28.817, -355]
  MoveL 4182 to (-19.54, 62.54, -174.33) mm, rotated rx 42.04 ry 15.1 rz -114.75 deg; joints [-15.607, -41.338, 105.241, 145.949, 50.041, -28.828, -355]
  MoveL 4183 to (-20.36, 62.66, -172.87) mm, rotated rx 42.04 ry 15.1 rz -114.75 deg; joints [-15.551, -41.394, 105.273, 146.005, 50.008, -28.837, -355]
  MoveL 4184 to (-23.91, 60.28, -172.87) mm, rotated rx 42.04 ry 15.1 rz -114.75 deg; joints [-15.57, -41.68, 105.553, 145.979, 50.008, -28.823, -355]
  MoveL 4185 to (-25.6, 59.15, -172.82) mm, rotated rx 42.04 ry 15.1 rz -114.75 deg; joints [-15.578, -41.817, 105.687, 145.968, 50.007, -28.817, -355]
  MoveL 4186 to (-27.25, 58.06, -172.73) mm, rotated rx 42.04 ry 15.1 rz -114.75 deg; joints [-15.583, -41.95, 105.817, 145.96, 50.005, -28.812, -355]
  MoveL 4187 to (-28.93, 56.94, -172.65) mm, rotated rx 42.04 ry 15.1 rz -114.75 deg; joints [-15.589, -42.086, 105.949, 145.951, 50.004, -28.807, -355]
  MoveL 4188 to (-30.57, 55.85, -172.55) mm, rotated rx 42.04 ry 15.1 rz -114.75 deg; joints [-15.594, -42.219, 106.079, 145.943, 50.002, -28.802, -355]
  MoveL 4189 to (-32.32, 54.71, -172.51) mm, rotated rx 42.04 ry 15.1 rz -114.75 deg; joints [-15.602, -42.36, 106.213, 145.931, 49.999, -28.793, -355]
  MoveL 4190 to (-34.21, 53.57, -172.47) mm, rotated rx 42.04 ry 15.1 rz -114.75 deg; joints [-15.611, -42.509, 106.349, 145.915, 49.99, -28.78, -355]
  MoveL 4191 to (-36.23, 52.1, -172.31) mm, rotated rx 42.04 ry 15.1 rz -114.75 deg; joints [-15.616, -42.677, 106.519, 145.909, 49.993, -28.779, -355]
  MoveL 4192 to (-38.1, 50.86, -172.06) mm, rotated rx 42.04 ry 15.1 rz -114.75 deg; joints [-15.617, -42.83, 106.668, 145.906, 49.99, -28.775, -355]
  MoveL 4193 to (-39.92, 49.64, -171.93) mm, rotated rx 42.04 ry 15.1 rz -114.75 deg; joints [-15.622, -42.978, 106.81, 145.897, 49.986, -28.769, -355]
  MoveL 4194 to (-41.69, 48.45, -171.69) mm, rotated rx 42.04 ry 15.1 rz -114.75 deg; joints [-15.623, -43.123, 106.951, 145.894, 49.983, -28.765, -355]
  MoveL 4195 to (-43.46, 47.25, -171.56) mm, rotated rx 42.04 ry 15.1 rz -114.75 deg; joints [-15.628, -43.268, 107.09, 145.886, 49.98, -28.759, -355]
  MoveL 4196 to (-45.23, 46.06, -171.45) mm, rotated rx 42.04 ry 15.1 rz -114.75 deg; joints [-15.633, -43.412, 107.229, 145.876, 49.976, -28.752, -355]
  MoveL 4197 to (-46.99, 44.85, -171.21) mm, rotated rx 42.04 ry 15.1 rz -114.75 deg; joints [-15.634, -43.557, 107.37, 145.873, 49.973, -28.748, -355]
  MoveL 4198 to (-48.75, 43.65, -171.09) mm, rotated rx 42.04 ry 15.1 rz -114.75 deg; joints [-15.639, -43.702, 107.508, 145.864, 49.969, -28.741, -355]
  MoveL 4199 to (-50.52, 42.45, -170.97) mm, rotated rx 42.04 ry 15.1 rz -114.75 deg; joints [-15.645, -43.846, 107.646, 145.854, 49.965, -28.734, -355]
  MoveL 4200 to (-52.28, 41.25, -170.85) mm, rotated rx 42.04 ry 15.1 rz -114.75 deg; joints [-15.65, -43.991, 107.784, 145.844, 49.961, -28.726, -355]
  MoveL 4201 to (-54.03, 40.02, -170.62) mm, rotated rx 42.04 ry 15.1 rz -114.75 deg; joints [-15.652, -44.136, 107.924, 145.841, 49.958, -28.723, -355]
  MoveL 4202 to (-55.79, 38.81, -170.51) mm, rotated rx 42.04 ry 15.1 rz -114.75 deg; joints [-15.658, -44.28, 108.062, 145.83, 49.953, -28.715, -355]
  MoveL 4203 to (-57.24, 37.77, -170.26) mm, rotated rx 42.04 ry 15.1 rz -114.75 deg; joints [-15.657, -44.402, 108.182, 145.831, 49.951, -28.714, -355]
  MoveL 4204 to (-58.57, 36.79, -169.94) mm, rotated rx 42.04 ry 15.1 rz -114.75 deg; joints [-15.652, -44.515, 108.296, 145.836, 49.951, -28.716, -355]
  MoveL 4205 to (-59.81, 35.83, -169.52) mm, rotated rx 42.04 ry 15.1 rz -114.75 deg; joints [-15.644, -44.624, 108.407, 145.848, 49.951, -28.722, -355]
  MoveL 4206 to (-58.1, 36.12, -168.56) mm, rotated rx 42.04 ry 15.1 rz -114.75 deg; joints [-15.604, -44.519, 108.369, 145.928, 49.996, -28.79, -355]
  MoveL 4207 to (-58.65, 35.8, -168.43) mm, rotated rx 42.04 ry 15.1 rz -114.75 deg; joints [-15.601, -44.563, 108.408, 145.928, 49.992, -28.788, -355]
  MoveL 4208 to (-59.18, 35.57, -168.35) mm, rotated rx 42.04 ry 15.1 rz -114.75 deg; joints [-15.6, -44.603, 108.439, 145.925, 49.984, -28.782, -355]
  MoveL 4209 to (-59.71, 35.46, -168.31) mm, rotated rx 42.04 ry 15.1 rz -114.75 deg; joints [-15.6, -44.638, 108.458, 145.918, 49.97, -28.77, -355]
  MoveL 4210 to (-60.24, 35.4, -168.3) mm, rotated rx 42.04 ry 15.1 rz -114.75 deg; joints [-15.6, -44.672, 108.472, 145.909, 49.955, -28.756, -355]
  MoveL 4211 to (-63.92, 35.37, -168.29) mm, rotated rx 42.04 ry 15.1 rz -114.75 deg; joints [-15.602, -44.891, 108.537, 145.833, 49.826, -28.641, -355]
  MoveL 4212 to (-64.38, 35.36, -168.28) mm, rotated rx 42.04 ry 15.1 rz -114.75 deg; joints [-15.602, -44.919, 108.545, 145.824, 49.811, -28.627, -355]
  MoveL 4213 to (-64.8, 35.34, -168.25) mm, rotated rx 42.04 ry 15.1 rz -114.75 deg; joints [-15.601, -44.945, 108.554, 145.817, 49.797, -28.615, -355]
  MoveL 4214 to (-65.28, 35.34, -168.24) mm, rotated rx 42.04 ry 15.1 rz -114.75 deg; joints [-15.601, -44.974, 108.563, 145.808, 49.78, -28.6, -355]
  MoveL 4215 to (-65.81, 35.33, -168.24) mm, rotated rx 42.04 ry 15.1 rz -114.75 deg; joints [-15.601, -45.005, 108.572, 145.797, 49.761, -28.584, -355]
  MoveL 4216 to (-67.38, 35.33, -168.24) mm, rotated rx 42.04 ry 15.1 rz -114.75 deg; joints [-15.602, -45.098, 108.598, 145.764, 49.706, -28.534, -355]
  MoveL 4217 to (-68.01, 35.32, -168.22) mm, rotated rx 42.04 ry 15.1 rz -114.75 deg; joints [-15.602, -45.136, 108.609, 145.752, 49.684, -28.515, -355]
  MoveL 4218 to (-68.72, 35.29, -168.18) mm, rotated rx 42.04 ry 15.1 rz -114.75 deg; joints [-15.601, -45.18, 108.624, 145.739, 49.66, -28.494, -355]
  MoveL 4219 to (-69.37, 35.27, -168.16) mm, rotated rx 42.04 ry 15.1 rz -114.75 deg; joints [-15.6, -45.219, 108.636, 145.727, 49.638, -28.474, -355]
  MoveL 4220 to (-70.42, 35.27, -168.16) mm, rotated rx 42.04 ry 15.1 rz -114.75 deg; joints [-15.601, -45.281, 108.653, 145.704, 49.601, -28.441, -355]
  MoveL 4221 to (-71.86, 35.34, -168.24) mm, rotated rx 42.04 ry 15.1 rz -114.75 deg; joints [-15.604, -45.363, 108.669, 145.668, 49.546, -28.389, -355]
  MoveL 4222 to (-73.03, 35.55, -168.5) mm, rotated rx 42.04 ry 15.1 rz -114.75 deg; joints [-15.613, -45.424, 108.665, 145.626, 49.496, -28.337, -355]
  MoveL 4223 to (-73.92, 35.9, -168.92) mm, rotated rx 42.04 ry 15.1 rz -114.75 deg; joints [-15.627, -45.462, 108.642, 145.58, 49.449, -28.285, -355]
  MoveL 4224 to (-74.26, 36.12, -169.19) mm, rotated rx 42.04 ry 15.1 rz -114.75 deg; joints [-15.637, -45.472, 108.623, 145.554, 49.427, -28.259, -355]
  MoveL 4225 to (-74.53, 36.38, -169.5) mm, rotated rx 42.04 ry 15.1 rz -114.75 deg; joints [-15.647, -45.477, 108.6, 145.528, 49.406, -28.232, -355]
  MoveL 4226 to (-74.85, 37, -170.26) mm, rotated rx 42.04 ry 15.1 rz -114.75 deg; joints [-15.672, -45.47, 108.538, 145.471, 49.367, -28.179, -355]
  MoveL 4227 to (-74.9, 37.76, -171.18) mm, rotated rx 42.04 ry 15.1 rz -114.75 deg; joints [-15.702, -45.441, 108.456, 145.409, 49.332, -28.125, -355]
  MoveL 4228 to (-74.16, 39.7, -173.54) mm, rotated rx 42.04 ry 15.1 rz -114.75 deg; joints [-15.778, -45.315, 108.236, 145.271, 49.273, -28.017, -355]
  MoveL 4229 to (-72.63, 41.58, -175.89) mm, rotated rx 42.04 ry 15.1 rz -114.75 deg; joints [-15.854, -45.145, 108.006, 145.15, 49.245, -27.935, -355]
  MoveL 4230 to (-70.63, 42.81, -177.57) mm, rotated rx 42.04 ry 15.1 rz -114.75 deg; joints [-15.908, -44.974, 107.838, 145.085, 49.261, -27.91, -355]
  MoveL 4231 to (-69.46, 43.18, -178.16) mm, rotated rx 42.04 ry 15.1 rz -114.75 deg; joints [-15.927, -44.888, 107.776, 145.074, 49.286, -27.919, -355]
  MoveL 4232 to (-68.17, 43.38, -178.58) mm, rotated rx 42.04 ry 15.1 rz -114.75 deg; joints [-15.941, -44.802, 107.73, 145.077, 49.322, -27.942, -355]
  MoveL 4233 to (-65.26, 43.3, -178.91) mm, rotated rx 42.04 ry 15.1 rz -114.75 deg; joints [-15.953, -44.631, 107.683, 145.123, 49.427, -28.03, -355]
  MoveL 4234 to (-62.14, 42.9, -178.91) mm, rotated rx 42.04 ry 15.1 rz -114.75 deg; joints [-15.954, -44.461, 107.667, 145.197, 49.554, -28.145, -355]
  MoveL 4235 to (-61.16, 42.82, -178.96) mm, rotated rx 42.04 ry 15.1 rz -114.75 deg; joints [-15.956, -44.405, 107.656, 145.216, 49.592, -28.178, -355]
  MoveL 4236 to (-60.64, 42.75, -178.96) mm, rotated rx 42.04 ry 15.1 rz -114.75 deg; joints [-15.957, -44.377, 107.654, 145.228, 49.613, -28.197, -355]
  MoveL 4237 to (-60.11, 42.69, -178.96) mm, rotated rx 42.04 ry 15.1 rz -114.75 deg; joints [-15.957, -44.347, 107.65, 145.241, 49.634, -28.216, -355]
  MoveL 4238 to (-59.54, 42.63, -178.99) mm, rotated rx 42.04 ry 15.1 rz -114.75 deg; joints [-15.958, -44.316, 107.646, 145.253, 49.656, -28.236, -355]
  MoveL 4239 to (-58.9, 42.58, -179.05) mm, rotated rx 42.04 ry 15.1 rz -114.75 deg; joints [-15.96, -44.279, 107.638, 145.264, 49.681, -28.256, -355]
  MoveL 4240 to (-58.32, 42.53, -179.08) mm, rotated rx 42.04 ry 15.1 rz -114.75 deg; joints [-15.961, -44.246, 107.632, 145.275, 49.703, -28.276, -355]
  MoveL 4241 to (-57.8, 42.47, -179.09) mm, rotated rx 42.04 ry 15.1 rz -114.75 deg; joints [-15.962, -44.217, 107.628, 145.286, 49.724, -28.294, -355]
  MoveL 4242 to (-57.32, 42.43, -179.12) mm, rotated rx 42.04 ry 15.1 rz -114.75 deg; joints [-15.963, -44.19, 107.623, 145.296, 49.742, -28.31, -355]
  MoveL 4243 to (-56.87, 42.41, -179.17) mm, rotated rx 42.04 ry 15.1 rz -114.75 deg; joints [-15.965, -44.163, 107.616, 145.303, 49.759, -28.324, -355]
  MoveL 4244 to (-56.41, 42.38, -179.21) mm, rotated rx 42.04 ry 15.1 rz -114.75 deg; joints [-15.967, -44.137, 107.61, 145.311, 49.776, -28.338, -355]
  MoveL 4245 to (-55.9, 42.32, -179.22) mm, rotated rx 42.04 ry 15.1 rz -114.75 deg; joints [-15.967, -44.109, 107.606, 145.322, 49.796, -28.356, -355]
  MoveL 4246 to (-55.39, 42.27, -179.22) mm, rotated rx 42.04 ry 15.1 rz -114.75 deg; joints [-15.968, -44.08, 107.602, 145.333, 49.816, -28.374, -355]
  MoveL 4247 to (-54.88, 42.24, -179.23) mm, rotated rx 42.04 ry 15.1 rz -114.75 deg; joints [-15.968, -44.051, 107.595, 145.344, 49.835, -28.391, -355]
  MoveL 4248 to (-54.39, 42.26, -179.25) mm, rotated rx 42.04 ry 15.1 rz -114.75 deg; joints [-15.968, -44.021, 107.584, 145.353, 49.851, -28.405, -355]
  MoveL 4249 to (-53.92, 42.34, -179.28) mm, rotated rx 42.04 ry 15.1 rz -114.75 deg; joints [-15.968, -43.991, 107.569, 145.359, 49.863, -28.416, -355]
  MoveL 4250 to (-53.49, 42.48, -179.33) mm, rotated rx 42.04 ry 15.1 rz -114.75 deg; joints [-15.969, -43.96, 107.548, 145.364, 49.871, -28.423, -355]
  MoveL 4251 to (-53.06, 42.65, -179.37) mm, rotated rx 42.04 ry 15.1 rz -114.75 deg; joints [-15.969, -43.929, 107.525, 145.367, 49.878, -28.429, -355]
  MoveL 4252 to (-54.55, 42.33, -180.34) mm, rotated rx 42.04 ry 15.1 rz -114.75 deg; joints [-16.01, -44.02, 107.562, 145.292, 49.844, -28.369, -355]
  MoveL 4253 to (-53.1, 43.24, -180.72) mm, rotated rx 42.04 ry 15.1 rz -114.75 deg; joints [-16.016, -43.902, 107.45, 145.288, 49.851, -28.371, -355]
  MoveL 4254 to (-51.53, 44.15, -181) mm, rotated rx 42.04 ry 15.1 rz -114.75 deg; joints [-16.019, -43.777, 107.338, 145.29, 49.862, -28.379, -355]
  MoveL 4255 to (-49.83, 45.09, -181.2) mm, rotated rx 42.04 ry 15.1 rz -114.75 deg; joints [-16.018, -43.644, 107.223, 145.299, 49.877, -28.392, -355]
  MoveL 4256 to (-47.94, 46.09, -181.42) mm, rotated rx 42.04 ry 15.1 rz -114.75 deg; joints [-16.018, -43.498, 107.099, 145.31, 49.894, -28.408, -355]
  MoveL 4257 to (-46.04, 47.06, -181.54) mm, rotated rx 42.04 ry 15.1 rz -114.75 deg; joints [-16.014, -43.354, 106.978, 145.326, 49.913, -28.428, -355]
  MoveL 4258 to (-44.13, 48.02, -181.65) mm, rotated rx 42.04 ry 15.1 rz -114.75 deg; joints [-16.01, -43.209, 106.857, 145.343, 49.931, -28.448, -355]
  MoveL 4259 to (-42.23, 49.01, -181.88) mm, rotated rx 42.04 ry 15.1 rz -114.75 deg; joints [-16.01, -43.063, 106.732, 145.353, 49.949, -28.464, -355]
  MoveL 4260 to (-40.33, 49.97, -182) mm, rotated rx 42.04 ry 15.1 rz -114.75 deg; joints [-16.006, -42.918, 106.611, 145.369, 49.967, -28.483, -355]
  MoveL 4261 to (-38.42, 50.93, -182.12) mm, rotated rx 42.04 ry 15.1 rz -114.75 deg; joints [-16.002, -42.773, 106.489, 145.385, 49.985, -28.502, -355]
  MoveL 4262 to (-36.52, 51.9, -182.36) mm, rotated rx 42.04 ry 15.1 rz -114.75 deg; joints [-16.003, -42.628, 106.365, 145.394, 50.002, -28.517, -355]
  MoveL 4263 to (-34.61, 52.85, -182.48) mm, rotated rx 42.04 ry 15.1 rz -114.75 deg; joints [-15.999, -42.483, 106.243, 145.41, 50.02, -28.536, -355]
  MoveL 4264 to (-32.7, 53.81, -182.6) mm, rotated rx 42.04 ry 15.1 rz -114.75 deg; joints [-15.995, -42.338, 106.121, 145.425, 50.038, -28.555, -355]
  MoveL 4265 to (-30.9, 54.7, -182.79) mm, rotated rx 42.04 ry 15.1 rz -114.75 deg; joints [-15.994, -42.201, 106.004, 145.435, 50.055, -28.57, -355]
  MoveL 4266 to (-29.26, 55.51, -183) mm, rotated rx 42.04 ry 15.1 rz -114.75 deg; joints [-15.995, -42.077, 105.898, 145.443, 50.07, -28.583, -355]
  MoveL 4267 to (-27.5, 56.38, -183.11) mm, rotated rx 42.04 ry 15.1 rz -114.75 deg; joints [-15.992, -41.944, 105.785, 145.457, 50.086, -28.6, -355]
  MoveL 4268 to (-25.6, 57.43, -183.11) mm, rotated rx 42.04 ry 15.1 rz -114.75 deg; joints [-15.983, -41.798, 105.655, 145.476, 50.097, -28.616, -355]
  MoveL 4269 to (-23.15, 58.62, -183.2) mm, rotated rx 42.04 ry 15.1 rz -114.75 deg; joints [-15.975, -41.614, 105.501, 145.498, 50.119, -28.641, -355]
  MoveL 4270 to (-20.89, 59.6, -183.44) mm, rotated rx 42.04 ry 15.1 rz -114.75 deg; joints [-15.976, -41.447, 105.365, 145.512, 50.145, -28.664, -355]
  MoveL 4271 to (-19.06, 60.49, -183.62) mm, rotated rx 42.04 ry 15.1 rz -114.75 deg; joints [-15.975, -41.309, 105.247, 145.523, 50.161, -28.679, -355]
  MoveL 4272 to (-17.37, 61.29, -183.94) mm, rotated rx 42.04 ry 15.1 rz -114.75 deg; joints [-15.98, -41.181, 105.137, 145.525, 50.177, -28.69, -355]
  MoveL 4273 to (-15.52, 62.17, -184.12) mm, rotated rx 42.04 ry 15.1 rz -114.75 deg; joints [-15.979, -41.042, 105.018, 145.536, 50.194, -28.705, -355]
  MoveL 4274 to (-13.73, 63, -184.32) mm, rotated rx 42.04 ry 15.1 rz -114.75 deg; joints [-15.979, -40.908, 104.904, 145.545, 50.21, -28.72, -355]
  MoveL 4275 to (-11.98, 63.79, -184.6) mm, rotated rx 42.04 ry 15.1 rz -114.75 deg; joints [-15.983, -40.777, 104.793, 145.55, 50.228, -28.733, -355]
  MoveL 4276 to (-11.08, 63.63, -185.37) mm, rotated rx 42.04 ry 15.1 rz -114.75 deg; joints [-16.013, -40.724, 104.775, 145.531, 50.264, -28.745, -355]
  MoveL 4277 to (-11.29, 63.31, -185.75) mm, rotated rx 42.04 ry 15.1 rz -114.75 deg; joints [-16.03, -40.743, 104.8, 145.513, 50.273, -28.741, -355]
  MoveL 4278 to (-11.31, 63.23, -185.99) mm, rotated rx 42.04 ry 15.1 rz -114.75 deg; joints [-16.04, -40.745, 104.803, 145.502, 50.276, -28.737, -355]
  MoveL 4279 to (-11.16, 63.38, -186.12) mm, rotated rx 42.04 ry 15.1 rz -114.75 deg; joints [-16.043, -40.731, 104.785, 145.496, 50.274, -28.732, -355]
  MoveL 4280 to (-10.85, 63.81, -186.17) mm, rotated rx 42.04 ry 15.1 rz -114.75 deg; joints [-16.042, -40.698, 104.74, 145.492, 50.263, -28.724, -355]
  MoveL 4281 to (-10.48, 64.36, -186.2) mm, rotated rx 42.04 ry 15.1 rz -114.75 deg; joints [-16.039, -40.658, 104.682, 145.487, 50.248, -28.712, -355]
  MoveL 4282 to (-9.7, 65.73, -186.2) mm, rotated rx 42.04 ry 15.1 rz -114.75 deg; joints [-16.028, -40.569, 104.545, 145.478, 50.206, -28.683, -355]
  MoveL 4283 to (-9.42, 66.2, -186.21) mm, rotated rx 42.04 ry 15.1 rz -114.75 deg; joints [-16.024, -40.537, 104.498, 145.474, 50.192, -28.672, -355]
  MoveL 4284 to (-9.14, 66.66, -186.24) mm, rotated rx 42.04 ry 15.1 rz -114.75 deg; joints [-16.021, -40.506, 104.451, 145.47, 50.179, -28.662, -355]
  MoveL 4285 to (-8.84, 67.12, -186.29) mm, rotated rx 42.04 ry 15.1 rz -114.75 deg; joints [-16.02, -40.473, 104.403, 145.465, 50.166, -28.652, -355]
  MoveL 4286 to (-8.52, 67.57, -186.36) mm, rotated rx 42.04 ry 15.1 rz -114.75 deg; joints [-16.019, -40.439, 104.355, 145.46, 50.154, -28.642, -355]
  MoveL 4287 to (-8.21, 68.03, -186.42) mm, rotated rx 42.04 ry 15.1 rz -114.75 deg; joints [-16.017, -40.405, 104.307, 145.454, 50.141, -28.632, -355]
  MoveL 4288 to (-7.95, 68.46, -186.44) mm, rotated rx 42.04 ry 15.1 rz -114.75 deg; joints [-16.015, -40.376, 104.263, 145.451, 50.129, -28.622, -355]
  MoveL 4289 to (-7.72, 68.85, -186.46) mm, rotated rx 42.04 ry 15.1 rz -114.75 deg; joints [-16.012, -40.35, 104.223, 145.447, 50.117, -28.614, -355]
  MoveL 4290 to (-6.94, 70.21, -186.46) mm, rotated rx 42.04 ry 15.1 rz -114.75 deg; joints [-16.001, -40.26, 104.086, 145.438, 50.075, -28.584, -355]
  MoveL 4291 to (-6.67, 70.66, -186.47) mm, rotated rx 42.04 ry 15.1 rz -114.75 deg; joints [-15.998, -40.23, 104.04, 145.434, 50.062, -28.574, -355]
  MoveL 4292 to (-6.42, 71.06, -186.5) mm, rotated rx 42.04 ry 15.1 rz -114.75 deg; joints [-15.996, -40.202, 103.998, 145.43, 50.05, -28.565, -355]
  MoveL 4293 to (-6.16, 71.43, -186.55) mm, rotated rx 42.04 ry 15.1 rz -114.75 deg; joints [-15.995, -40.174, 103.96, 145.426, 50.04, -28.557, -355]
  MoveL 4294 to (-5.92, 71.81, -186.59) mm, rotated rx 42.04 ry 15.1 rz -114.75 deg; joints [-15.993, -40.147, 103.92, 145.422, 50.03, -28.548, -355]
  MoveL 4295 to (-5.66, 72.22, -186.6) mm, rotated rx 42.04 ry 15.1 rz -114.75 deg; joints [-15.991, -40.119, 103.877, 145.419, 50.017, -28.539, -355]
  MoveL 4296 to (-5.4, 72.68, -186.6) mm, rotated rx 42.04 ry 15.1 rz -114.75 deg; joints [-15.987, -40.089, 103.831, 145.415, 50.003, -28.529, -355]
  MoveL 4297 to (-3.7, 75.07, -186.94) mm, rotated rx 42.04 ry 15.1 rz -114.75 deg; joints [-15.981, -39.909, 103.576, 145.387, 49.939, -28.476, -355]
  MoveL 4298 to (-2.76, 75.98, -187.36) mm, rotated rx 42.04 ry 15.1 rz -114.75 deg; joints [-15.989, -39.821, 103.467, 145.367, 49.924, -28.456, -355]
  MoveL 4299 to (-1.75, 76.71, -187.95) mm, rotated rx 42.04 ry 15.1 rz -114.75 deg; joints [-16.005, -39.733, 103.369, 145.343, 49.92, -28.441, -355]
  MoveL 4300 to (0.46, 77.61, -189.64) mm, rotated rx 42.04 ry 15.1 rz -114.75 deg; joints [-16.06, -39.562, 103.21, 145.282, 49.944, -28.424, -355]
  MoveL 4301 to (2.92, 77.77, -192) mm, rotated rx 42.04 ry 15.1 rz -114.75 deg; joints [-16.146, -39.394, 103.098, 145.206, 50.011, -28.424, -355]
  MoveL 4302 to (4.94, 77.27, -194.36) mm, rotated rx 42.04 ry 15.1 rz -114.75 deg; joints [-16.237, -39.274, 103.054, 145.133, 50.097, -28.438, -355]
  MoveL 4303 to (5.53, 76.8, -195.29) mm, rotated rx 42.04 ry 15.1 rz -114.75 deg; joints [-16.275, -39.247, 103.066, 145.105, 50.138, -28.449, -355]
  MoveL 4304 to (5.84, 76.19, -196.05) mm, rotated rx 42.04 ry 15.1 rz -114.75 deg; joints [-16.308, -39.243, 103.099, 145.084, 50.177, -28.461, -355]
  MoveL 4305 to (5.89, 75.83, -196.37) mm, rotated rx 42.04 ry 15.1 rz -114.75 deg; joints [-16.323, -39.249, 103.124, 145.075, 50.197, -28.469, -355]
  MoveL 4306 to (5.87, 75.43, -196.64) mm, rotated rx 42.04 ry 15.1 rz -114.75 deg; joints [-16.336, -39.261, 103.155, 145.068, 50.215, -28.476, -355]
  MoveL 4307 to (5.62, 74.52, -197.06) mm, rotated rx 42.04 ry 15.1 rz -114.75 deg; joints [-16.359, -39.302, 103.233, 145.059, 50.252, -28.493, -355]
  MoveL 4308 to (5.08, 73.48, -197.32) mm, rotated rx 42.04 ry 15.1 rz -114.75 deg; joints [-16.377, -39.365, 103.334, 145.055, 50.287, -28.513, -355]
  MoveL 4309 to (4.26, 72.28, -197.4) mm, rotated rx 42.04 ry 15.1 rz -114.75 deg; joints [-16.39, -39.451, 103.456, 145.057, 50.32, -28.534, -355]
  MoveL 4310 to (3.32, 71.03, -197.4) mm, rotated rx 42.04 ry 15.1 rz -114.75 deg; joints [-16.401, -39.547, 103.588, 145.062, 50.353, -28.556, -355]
  MoveL 4311 to (3, 70.61, -197.4) mm, rotated rx 42.04 ry 15.1 rz -114.75 deg; joints [-16.404, -39.579, 103.633, 145.063, 50.363, -28.564, -355]
  MoveL 4312 to (2.63, 70.17, -197.36) mm, rotated rx 42.04 ry 15.1 rz -114.75 deg; joints [-16.406, -39.615, 103.681, 145.066, 50.374, -28.571, -355]
  MoveL 4313 to (2.2, 69.68, -197.3) mm, rotated rx 42.04 ry 15.1 rz -114.75 deg; joints [-16.408, -39.656, 103.734, 145.07, 50.384, -28.58, -355]
  MoveL 4314 to (1.85, 69.24, -197.27) mm, rotated rx 42.04 ry 15.1 rz -114.75 deg; joints [-16.411, -39.691, 103.782, 145.072, 50.395, -28.587, -355]
  MoveL 4315 to (1.52, 68.82, -197.27) mm, rotated rx 42.04 ry 15.1 rz -114.75 deg; joints [-16.414, -39.724, 103.826, 145.074, 50.406, -28.595, -355]
  MoveL 4316 to (1.21, 68.41, -197.26) mm, rotated rx 42.04 ry 15.1 rz -114.75 deg; joints [-16.417, -39.756, 103.869, 145.076, 50.416, -28.602, -355]
  MoveL 4317 to (0.87, 68.03, -197.21) mm, rotated rx 42.04 ry 15.1 rz -114.75 deg; joints [-16.419, -39.788, 103.912, 145.079, 50.424, -28.609, -355]
  MoveL 4318 to (0.53, 67.66, -197.13) mm, rotated rx 42.04 ry 15.1 rz -114.75 deg; joints [-16.419, -39.821, 103.953, 145.083, 50.432, -28.615, -355]
  MoveL 4319 to (0.18, 67.3, -197.04) mm, rotated rx 42.04 ry 15.1 rz -114.75 deg; joints [-16.418, -39.854, 103.995, 145.087, 50.438, -28.622, -355]
  MoveL 4320 to (-0.17, 66.92, -196.97) mm, rotated rx 42.04 ry 15.1 rz -114.75 deg; joints [-16.419, -39.887, 104.037, 145.091, 50.446, -28.628, -355]
  MoveL 4321 to (-0.51, 66.51, -196.94) mm, rotated rx 42.04 ry 15.1 rz -114.75 deg; joints [-16.421, -39.92, 104.081, 145.094, 50.456, -28.635, -355]
  MoveL 4322 to (-0.83, 66.1, -196.92) mm, rotated rx 42.04 ry 15.1 rz -114.75 deg; joints [-16.424, -39.952, 104.125, 145.096, 50.466, -28.642, -355]
  MoveL 4323 to (-2.4, 64.09, -196.92) mm, rotated rx 42.04 ry 15.1 rz -114.75 deg; joints [-16.441, -40.109, 104.337, 145.102, 50.515, -28.676, -355]
  MoveL 4324 to (-2.68, 63.82, -196.89) mm, rotated rx 42.04 ry 15.1 rz -114.75 deg; joints [-16.442, -40.134, 104.367, 145.102, 50.519, -28.679, -355]
  MoveL 4325 to (-2.82, 63.72, -196.78) mm, rotated rx 42.04 ry 15.1 rz -114.75 deg; joints [-16.439, -40.146, 104.38, 145.107, 50.52, -28.681, -355]
  MoveL 4326 to (-2.76, 63.79, -196.55) mm, rotated rx 42.04 ry 15.1 rz -114.75 deg; joints [-16.429, -40.143, 104.378, 145.119, 50.519, -28.687, -355]
  MoveL 4327 to (-2.47, 64.01, -196.19) mm, rotated rx 42.04 ry 15.1 rz -114.75 deg; joints [-16.414, -40.122, 104.359, 145.139, 50.517, -28.696, -355]
  MoveL 4328 to (-3.22, 64.19, -195.45) mm, rotated rx 42.04 ry 15.1 rz -114.75 deg; joints [-16.385, -40.165, 104.373, 145.159, 50.485, -28.686, -355]
  MoveL 4329 to (-5.22, 63.5, -195.43) mm, rotated rx 42.04 ry 15.1 rz -114.75 deg; joints [-16.391, -40.306, 104.477, 145.134, 50.456, -28.656, -355]
  MoveL 4330 to (-7.3, 62.82, -195.3) mm, rotated rx 42.04 ry 15.1 rz -114.75 deg; joints [-16.393, -40.452, 104.583, 145.114, 50.424, -28.627, -355]
  MoveL 4331 to (-9.47, 62.15, -195.04) mm, rotated rx 42.04 ry 15.1 rz -114.75 deg; joints [-16.389, -40.604, 104.693, 145.098, 50.389, -28.597, -355]
  MoveL 4332 to (-11.48, 61.49, -194.91) mm, rotated rx 42.04 ry 15.1 rz -114.75 deg; joints [-16.391, -40.745, 104.796, 145.078, 50.358, -28.568, -355]
  MoveL 4333 to (-13.43, 60.86, -194.65) mm, rotated rx 42.04 ry 15.1 rz -114.75 deg; joints [-16.387, -40.882, 104.896, 145.065, 50.327, -28.542, -355]
  MoveL 4334 to (-15.44, 60.23, -194.29) mm, rotated rx 42.04 ry 15.1 rz -114.75 deg; joints [-16.38, -41.024, 105, 145.056, 50.294, -28.518, -355]
  MoveL 4335 to (-17.47, 59.54, -194.15) mm, rotated rx 42.04 ry 15.1 rz -114.75 deg; joints [-16.381, -41.167, 105.104, 145.036, 50.262, -28.488, -355]
  MoveL 4336 to (-19.48, 58.86, -194.05) mm, rotated rx 42.04 ry 15.1 rz -114.75 deg; joints [-16.384, -41.308, 105.207, 145.014, 50.231, -28.458, -355]
  MoveL 4337 to (-21.51, 58.17, -193.9) mm, rotated rx 42.04 ry 15.1 rz -114.75 deg; joints [-16.385, -41.451, 105.311, 144.994, 50.2, -28.428, -355]
  MoveL 4338 to (-23.5, 57.52, -193.62) mm, rotated rx 42.04 ry 15.1 rz -114.75 deg; joints [-16.38, -41.592, 105.413, 144.981, 50.167, -28.401, -355]
  MoveL 4339 to (-25.55, 56.78, -193.28) mm, rotated rx 42.04 ry 15.1 rz -114.75 deg; joints [-16.374, -41.74, 105.525, 144.971, 50.136, -28.378, -355]
  MoveL 4340 to (-27.55, 56.07, -193.1) mm, rotated rx 42.04 ry 15.1 rz -114.75 deg; joints [-16.374, -41.882, 105.63, 144.953, 50.105, -28.349, -355]
  MoveL 4341 to (-29.58, 55.37, -192.99) mm, rotated rx 42.04 ry 15.1 rz -114.75 deg; joints [-16.377, -42.025, 105.733, 144.931, 50.073, -28.318, -355]
  MoveL 4342 to (-31.58, 54.67, -192.91) mm, rotated rx 42.04 ry 15.1 rz -114.75 deg; joints [-16.381, -42.167, 105.834, 144.907, 50.042, -28.286, -355]
  MoveL 4343 to (-33.6, 53.94, -192.69) mm, rotated rx 42.04 ry 15.1 rz -114.75 deg; joints [-16.379, -42.311, 105.941, 144.89, 50.01, -28.258, -355]
  MoveL 4344 to (-35.6, 53.23, -192.56) mm, rotated rx 42.04 ry 15.1 rz -114.75 deg; joints [-16.381, -42.453, 106.043, 144.869, 49.978, -28.228, -355]
  MoveL 4345 to (-37.62, 52.52, -192.48) mm, rotated rx 42.04 ry 15.1 rz -114.75 deg; joints [-16.385, -42.596, 106.145, 144.845, 49.946, -28.195, -355]
  MoveL 4346 to (-39.61, 51.78, -192.25) mm, rotated rx 42.04 ry 15.1 rz -114.75 deg; joints [-16.383, -42.739, 106.251, 144.828, 49.915, -28.168, -355]
  MoveL 4347 to (-41.63, 51.03, -192.02) mm, rotated rx 42.04 ry 15.1 rz -114.75 deg; joints [-16.382, -42.885, 106.359, 144.812, 49.883, -28.14, -355]
  MoveL 4348 to (-43.68, 50.28, -191.87) mm, rotated rx 42.04 ry 15.1 rz -114.75 deg; joints [-16.383, -43.031, 106.464, 144.791, 49.85, -28.109, -355]
  MoveL 4349 to (-45.43, 49.61, -191.74) mm, rotated rx 42.04 ry 15.1 rz -114.75 deg; joints [-16.385, -43.157, 106.557, 144.772, 49.824, -28.083, -355]
  MoveL 4350 to (-46.94, 48.96, -191.53) mm, rotated rx 42.04 ry 15.1 rz -114.75 deg; joints [-16.383, -43.269, 106.645, 144.763, 49.803, -28.066, -355]
  MoveL 4351 to (-48.23, 48.33, -191.21) mm, rotated rx 42.04 ry 15.1 rz -114.75 deg; joints [-16.376, -43.368, 106.729, 144.764, 49.79, -28.058, -355]
  MoveL 4352 to (-46.78, 48.59, -190.25) mm, rotated rx 42.04 ry 15.1 rz -114.75 deg; joints [-16.337, -43.281, 106.698, 144.838, 49.825, -28.118, -355]
  MoveL 4353 to (-47.25, 48.43, -190.25) mm, rotated rx 42.04 ry 15.1 rz -114.75 deg; joints [-16.338, -43.314, 106.72, 144.831, 49.817, -28.11, -355]
  MoveL 4354 to (-47.73, 48.31, -190.25) mm, rotated rx 42.04 ry 15.1 rz -114.75 deg; joints [-16.339, -43.347, 106.74, 144.824, 49.806, -28.1, -355]
  MoveL 4355 to (-48.26, 48.27, -190.22) mm, rotated rx 42.04 ry 15.1 rz -114.75 deg; joints [-16.339, -43.379, 106.753, 144.815, 49.79, -28.085, -355]
  MoveL 4356 to (-48.82, 48.29, -190.18) mm, rotated rx 42.04 ry 15.1 rz -114.75 deg; joints [-16.337, -43.412, 106.762, 144.805, 49.77, -28.068, -355]
  MoveL 4357 to (-49.43, 48.37, -190.13) mm, rotated rx 42.04 ry 15.1 rz -114.75 deg; joints [-16.335, -43.446, 106.767, 144.794, 49.746, -28.047, -355]
  MoveL 4358 to (-50, 48.49, -190.09) mm, rotated rx 42.04 ry 15.1 rz -114.75 deg; joints [-16.333, -43.476, 106.767, 144.782, 49.722, -28.026, -355]
  MoveL 4359 to (-50.54, 48.62, -190.07) mm, rotated rx 42.04 ry 15.1 rz -114.75 deg; joints [-16.332, -43.504, 106.766, 144.769, 49.697, -28.004, -355]
  MoveL 4360 to (-51.05, 48.75, -190.07) mm, rotated rx 42.04 ry 15.1 rz -114.75 deg; joints [-16.331, -43.529, 106.763, 144.756, 49.674, -27.983, -355]
  MoveL 4361 to (-51.56, 48.89, -190.07) mm, rotated rx 42.04 ry 15.1 rz -114.75 deg; joints [-16.33, -43.555, 106.761, 144.743, 49.651, -27.962, -355]
  MoveL 4362 to (-52.14, 49, -190.02) mm, rotated rx 42.04 ry 15.1 rz -114.75 deg; joints [-16.328, -43.585, 106.761, 144.731, 49.626, -27.941, -355]
  MoveL 4363 to (-52.79, 49.11, -189.94) mm, rotated rx 42.04 ry 15.1 rz -114.75 deg; joints [-16.324, -43.621, 106.765, 144.72, 49.599, -27.919, -355]
  MoveL 4364 to (-53.3, 49.21, -189.89) mm, rotated rx 42.04 ry 15.1 rz -114.75 deg; joints [-16.322, -43.648, 106.766, 144.71, 49.577, -27.9, -355]
  MoveL 4365 to (-53.71, 49.3, -189.86) mm, rotated rx 42.04 ry 15.1 rz -114.75 deg; joints [-16.32, -43.669, 106.765, 144.701, 49.559, -27.884, -355]
  MoveL 4366 to (-54.18, 49.42, -189.85) mm, rotated rx 42.04 ry 15.1 rz -114.75 deg; joints [-16.319, -43.693, 106.763, 144.69, 49.537, -27.865, -355]
  MoveL 4367 to (-54.68, 49.55, -189.85) mm, rotated rx 42.04 ry 15.1 rz -114.75 deg; joints [-16.318, -43.718, 106.761, 144.677, 49.514, -27.844, -355]
  MoveL 4368 to (-55.18, 49.67, -189.83) mm, rotated rx 42.04 ry 15.1 rz -114.75 deg; joints [-16.317, -43.743, 106.759, 144.666, 49.492, -27.824, -355]
  MoveL 4369 to (-55.66, 49.78, -189.81) mm, rotated rx 42.04 ry 15.1 rz -114.75 deg; joints [-16.315, -43.768, 106.758, 144.655, 49.471, -27.806, -355]
  MoveL 4370 to (-56.16, 49.9, -189.79) mm, rotated rx 42.04 ry 15.1 rz -114.75 deg; joints [-16.314, -43.794, 106.756, 144.643, 49.448, -27.785, -355]
  MoveL 4371 to (-58.7, 50.57, -189.79) mm, rotated rx 42.04 ry 15.1 rz -114.75 deg; joints [-16.31, -43.921, 106.741, 144.577, 49.331, -27.679, -355]
  MoveL 4372 to (-60.09, 51.01, -189.88) mm, rotated rx 42.04 ry 15.1 rz -114.75 deg; joints [-16.311, -43.987, 106.725, 144.535, 49.264, -27.616, -355]
  MoveL 4373 to (-61.18, 51.5, -190.13) mm, rotated rx 42.04 ry 15.1 rz -114.75 deg; joints [-16.317, -44.033, 106.696, 144.49, 49.205, -27.555, -355]
  MoveL 4374 to (-61.98, 52.04, -190.54) mm, rotated rx 42.04 ry 15.1 rz -114.75 deg; joints [-16.329, -44.058, 106.654, 144.442, 49.153, -27.497, -355]
  MoveL 4375 to (-62.49, 52.65, -191.13) mm, rotated rx 42.04 ry 15.1 rz -114.75 deg; joints [-16.347, -44.062, 106.598, 144.39, 49.109, -27.442, -355]
  MoveL 4376 to (-62.7, 53.31, -191.87) mm, rotated rx 42.04 ry 15.1 rz -114.75 deg; joints [-16.37, -44.047, 106.53, 144.335, 49.073, -27.39, -355]
  MoveL 4377 to (-62.62, 54.02, -192.79) mm, rotated rx 42.04 ry 15.1 rz -114.75 deg; joints [-16.399, -44.01, 106.448, 144.277, 49.044, -27.341, -355]
  MoveL 4378 to (-61.57, 55.63, -195.12) mm, rotated rx 42.04 ry 15.1 rz -114.75 deg; joints [-16.475, -43.877, 106.246, 144.15, 49.009, -27.25, -355]
  MoveL 4379 to (-59.76, 57.01, -197.47) mm, rotated rx 42.04 ry 15.1 rz -114.75 deg; joints [-16.552, -43.706, 106.05, 144.044, 49.009, -27.192, -355]
  MoveL 4380 to (-57.6, 57.72, -199.17) mm, rotated rx 42.04 ry 15.1 rz -114.75 deg; joints [-16.61, -43.543, 105.918, 143.99, 49.051, -27.188, -355]
  MoveL 4381 to (-56.4, 57.82, -199.79) mm, rotated rx 42.04 ry 15.1 rz -114.75 deg; joints [-16.631, -43.464, 105.877, 143.983, 49.087, -27.206, -355]
  MoveL 4382 to (-55.1, 57.75, -200.24) mm, rotated rx 42.04 ry 15.1 rz -114.75 deg; joints [-16.648, -43.387, 105.852, 143.989, 49.134, -27.238, -355]
  MoveL 4383 to (-52.26, 57.11, -200.67) mm, rotated rx 42.04 ry 15.1 rz -114.75 deg; joints [-16.668, -43.239, 105.851, 144.039, 49.258, -27.343, -355]
  MoveL 4384 to (-51.3, 56.8, -200.71) mm, rotated rx 42.04 ry 15.1 rz -114.75 deg; joints [-16.672, -43.193, 105.861, 144.063, 49.304, -27.384, -355]
  MoveL 4385 to (-48.87, 55.82, -200.71) mm, rotated rx 42.04 ry 15.1 rz -114.75 deg; joints [-16.678, -43.084, 105.904, 144.132, 49.429, -27.499, -355]
  MoveL 4386 to (-47.92, 55.48, -200.77) mm, rotated rx 42.04 ry 15.1 rz -114.75 deg; joints [-16.683, -43.039, 105.916, 144.155, 49.476, -27.541, -355]
  MoveL 4387 to (-46.95, 55.09, -200.77) mm, rotated rx 42.04 ry 15.1 rz -114.75 deg; joints [-16.685, -42.995, 105.934, 144.183, 49.527, -27.587, -355]
  MoveL 4388 to (-46.5, 54.91, -200.78) mm, rotated rx 42.04 ry 15.1 rz -114.75 deg; joints [-16.687, -42.974, 105.941, 144.195, 49.55, -27.607, -355]
  MoveL 4389 to (-46.09, 54.77, -200.8) mm, rotated rx 42.04 ry 15.1 rz -114.75 deg; joints [-16.688, -42.955, 105.946, 144.205, 49.57, -27.625, -355]
  MoveL 4390 to (-45.66, 54.6, -200.81) mm, rotated rx 42.04 ry 15.1 rz -114.75 deg; joints [-16.69, -42.935, 105.952, 144.216, 49.592, -27.645, -355]
  MoveL 4391 to (-43.23, 53.62, -200.82) mm, rotated rx 42.04 ry 15.1 rz -114.75 deg; joints [-16.697, -42.825, 105.994, 144.283, 49.717, -27.758, -355]
  MoveL 4392 to (-42.77, 53.45, -200.83) mm, rotated rx 42.04 ry 15.1 rz -114.75 deg; joints [-16.699, -42.803, 106, 144.295, 49.74, -27.778, -355]
  MoveL 4393 to (-42.32, 53.31, -200.87) mm, rotated rx 42.04 ry 15.1 rz -114.75 deg; joints [-16.701, -42.781, 106.003, 144.305, 49.761, -27.797, -355]
  MoveL 4394 to (-41.9, 53.22, -200.91) mm, rotated rx 42.04 ry 15.1 rz -114.75 deg; joints [-16.703, -42.759, 106.003, 144.313, 49.78, -27.812, -355]
  MoveL 4395 to (-41.47, 53.15, -200.95) mm, rotated rx 42.04 ry 15.1 rz -114.75 deg; joints [-16.705, -42.735, 106.001, 144.321, 49.797, -27.827, -355]
  MoveL 4396 to (-41.03, 53.15, -200.96) mm, rotated rx 42.04 ry 15.1 rz -114.75 deg; joints [-16.705, -42.709, 105.992, 144.33, 49.811, -27.841, -355]
  MoveL 4397 to (-40.58, 53.2, -200.97) mm, rotated rx 42.04 ry 15.1 rz -114.75 deg; joints [-16.704, -42.682, 105.98, 144.338, 49.824, -27.852, -355]
  MoveL 4398 to (-41.34, 53.26, -201.71) mm, rotated rx 42.04 ry 15.1 rz -114.75 deg; joints [-16.732, -42.719, 105.975, 144.283, 49.797, -27.807, -355]
  MoveL 4399 to (-40.01, 53.79, -202.26) mm, rotated rx 42.04 ry 15.1 rz -114.75 deg; joints [-16.748, -42.619, 105.893, 144.273, 49.816, -27.813, -355]
  MoveL 4400 to (-38.53, 54.28, -202.68) mm, rotated rx 42.04 ry 15.1 rz -114.75 deg; joints [-16.759, -42.512, 105.814, 144.274, 49.841, -27.829, -355]
  MoveL 4401 to (-36.83, 54.75, -202.99) mm, rotated rx 42.04 ry 15.1 rz -114.75 deg; joints [-16.766, -42.394, 105.735, 144.285, 49.875, -27.856, -355]
  MoveL 4402 to (-34.86, 55.21, -203.17) mm, rotated rx 42.04 ry 15.1 rz -114.75 deg; joints [-16.768, -42.262, 105.654, 144.307, 49.917, -27.894, -355]
  MoveL 4403 to (-32.82, 55.68, -203.37) mm, rotated rx 42.04 ry 15.1 rz -114.75 deg; joints [-16.771, -42.125, 105.57, 144.331, 49.961, -27.934, -355]
  MoveL 4404 to (-30.73, 56.13, -203.49) mm, rotated rx 42.04 ry 15.1 rz -114.75 deg; joints [-16.77, -41.986, 105.488, 144.359, 50.007, -27.977, -355]
  MoveL 4405 to (-28.65, 56.6, -203.71) mm, rotated rx 42.04 ry 15.1 rz -114.75 deg; joints [-16.774, -41.847, 105.403, 144.381, 50.051, -28.016, -355]
  MoveL 4406 to (-26.56, 57.04, -203.83) mm, rotated rx 42.04 ry 15.1 rz -114.75 deg; joints [-16.773, -41.708, 105.321, 144.41, 50.097, -28.059, -355]
  MoveL 4407 to (-24.48, 57.49, -203.95) mm, rotated rx 42.04 ry 15.1 rz -114.75 deg; joints [-16.773, -41.57, 105.238, 144.437, 50.142, -28.102, -355]
  MoveL 4408 to (-22.39, 57.93, -204.06) mm, rotated rx 42.04 ry 15.1 rz -114.75 deg; joints [-16.772, -41.432, 105.156, 144.465, 50.188, -28.144, -355]
  MoveL 4409 to (-20.3, 58.38, -204.3) mm, rotated rx 42.04 ry 15.1 rz -114.75 deg; joints [-16.776, -41.292, 105.071, 144.486, 50.233, -28.183, -355]
  MoveL 4410 to (-18.21, 58.81, -204.42) mm, rotated rx 42.04 ry 15.1 rz -114.75 deg; joints [-16.776, -41.154, 104.988, 144.514, 50.278, -28.225, -355]
  MoveL 4411 to (-16.22, 59.29, -204.52) mm, rotated rx 42.04 ry 15.1 rz -114.75 deg; joints [-16.774, -41.02, 104.903, 144.539, 50.317, -28.263, -355]
  MoveL 4412 to (-14.29, 59.87, -204.73) mm, rotated rx 42.04 ry 15.1 rz -114.75 deg; joints [-16.776, -40.886, 104.809, 144.556, 50.35, -28.292, -355]
  MoveL 4413 to (-11.83, 60.35, -204.87) mm, rotated rx 42.04 ry 15.1 rz -114.75 deg; joints [-16.776, -40.724, 104.713, 144.587, 50.404, -28.342, -355]
  MoveL 4414 to (-9.41, 60.7, -204.95) mm, rotated rx 42.04 ry 15.1 rz -114.75 deg; joints [-16.775, -40.569, 104.63, 144.623, 50.462, -28.396, -355]
  MoveL 4415 to (-7.15, 61.09, -204.98) mm, rotated rx 42.04 ry 15.1 rz -114.75 deg; joints [-16.772, -40.423, 104.547, 144.658, 50.513, -28.446, -355]
  MoveL 4416 to (-5.14, 61.5, -205.03) mm, rotated rx 42.04 ry 15.1 rz -114.75 deg; joints [-16.769, -40.291, 104.469, 144.686, 50.556, -28.487, -355]
  MoveL 4417 to (-3.22, 61.89, -205.15) mm, rotated rx 42.04 ry 15.1 rz -114.75 deg; joints [-16.769, -40.164, 104.391, 144.71, 50.596, -28.524, -355]
  MoveL 4418 to (-1.23, 62.3, -205.21) mm, rotated rx 42.04 ry 15.1 rz -114.75 deg; joints [-16.767, -40.033, 104.311, 144.736, 50.637, -28.563, -355]
  MoveL 4419 to (0.85, 62.72, -205.28) mm, rotated rx 42.04 ry 15.1 rz -114.75 deg; joints [-16.765, -39.896, 104.227, 144.764, 50.681, -28.604, -355]
  MoveL 4420 to (2.8, 63.09, -205.46) mm, rotated rx 42.04 ry 15.1 rz -114.75 deg; joints [-16.767, -39.767, 104.148, 144.784, 50.722, -28.64, -355]
  MoveL 4421 to (4.68, 63.43, -205.78) mm, rotated rx 42.04 ry 15.1 rz -114.75 deg; joints [-16.775, -39.643, 104.071, 144.797, 50.763, -28.671, -355]
  MoveL 4422 to (5.49, 63.13, -206.82) mm, rotated rx 42.04 ry 15.1 rz -114.75 deg; joints [-16.816, -39.595, 104.059, 144.765, 50.801, -28.679, -355]
  MoveL 4423 to (5.26, 63.03, -207.34) mm, rotated rx 42.04 ry 15.1 rz -114.75 deg; joints [-16.837, -39.609, 104.063, 144.736, 50.799, -28.663, -355]
  MoveL 4424 to (5.25, 63, -207.66) mm, rotated rx 42.04 ry 15.1 rz -114.75 deg; joints [-16.849, -39.607, 104.059, 144.72, 50.8, -28.655, -355]
  MoveL 4425 to (5.46, 63.06, -207.82) mm, rotated rx 42.04 ry 15.1 rz -114.75 deg; joints [-16.855, -39.592, 104.046, 144.715, 50.804, -28.654, -355]
  MoveL 4426 to (5.84, 63.24, -207.86) mm, rotated rx 42.04 ry 15.1 rz -114.75 deg; joints [-16.854, -39.563, 104.021, 144.717, 50.806, -28.657, -355]
  MoveL 4427 to (6.28, 63.52, -207.87) mm, rotated rx 42.04 ry 15.1 rz -114.75 deg; joints [-16.852, -39.528, 103.986, 144.72, 50.806, -28.658, -355]
  MoveL 4428 to (6.74, 63.9, -207.89) mm, rotated rx 42.04 ry 15.1 rz -114.75 deg; joints [-16.849, -39.489, 103.942, 144.721, 50.802, -28.656, -355]
  MoveL 4429 to (7.21, 64.32, -207.9) mm, rotated rx 42.04 ry 15.1 rz -114.75 deg; joints [-16.846, -39.448, 103.895, 144.722, 50.795, -28.652, -355]
  MoveL 4430 to (9.77, 66.94, -207.9) mm, rotated rx 42.04 ry 15.1 rz -114.75 deg; joints [-16.823, -39.214, 103.605, 144.723, 50.745, -28.622, -355]
  MoveL 4431 to (10.09, 67.25, -207.92) mm, rotated rx 42.04 ry 15.1 rz -114.75 deg; joints [-16.822, -39.185, 103.571, 144.722, 50.74, -28.618, -355]
  MoveL 4432 to (10.43, 67.59, -207.93) mm, rotated rx 42.04 ry 15.1 rz -114.75 deg; joints [-16.819, -39.154, 103.532, 144.722, 50.733, -28.614, -355]
  MoveL 4433 to (10.8, 67.96, -207.94) mm, rotated rx 42.04 ry 15.1 rz -114.75 deg; joints [-16.816, -39.12, 103.491, 144.722, 50.726, -28.61, -355]
  MoveL 4434 to (11.16, 68.3, -207.96) mm, rotated rx 42.04 ry 15.1 rz -114.75 deg; joints [-16.814, -39.088, 103.453, 144.721, 50.72, -28.606, -355]
  MoveL 4435 to (11.5, 68.61, -208) mm, rotated rx 42.04 ry 15.1 rz -114.75 deg; joints [-16.812, -39.058, 103.416, 144.72, 50.715, -28.602, -355]
  MoveL 4436 to (11.83, 68.89, -208.06) mm, rotated rx 42.04 ry 15.1 rz -114.75 deg; joints [-16.812, -39.029, 103.383, 144.719, 50.711, -28.599, -355]
  MoveL 4437 to (12.18, 69.21, -208.09) mm, rotated rx 42.04 ry 15.1 rz -114.75 deg; joints [-16.811, -38.998, 103.346, 144.718, 50.706, -28.595, -355]
  MoveL 4438 to (12.53, 69.55, -208.11) mm, rotated rx 42.04 ry 15.1 rz -114.75 deg; joints [-16.808, -38.967, 103.308, 144.717, 50.7, -28.591, -355]
  MoveL 4439 to (12.88, 69.9, -208.11) mm, rotated rx 42.04 ry 15.1 rz -114.75 deg; joints [-16.805, -38.934, 103.268, 144.717, 50.693, -28.587, -355]
  MoveL 4440 to (13.25, 70.28, -208.11) mm, rotated rx 42.04 ry 15.1 rz -114.75 deg; joints [-16.802, -38.901, 103.227, 144.717, 50.686, -28.583, -355]
  MoveL 4441 to (15.49, 72.15, -208.46) mm, rotated rx 42.04 ry 15.1 rz -114.75 deg; joints [-16.798, -38.707, 103.002, 144.707, 50.66, -28.562, -355]
  MoveL 4442 to (16.62, 72.79, -208.89) mm, rotated rx 42.04 ry 15.1 rz -114.75 deg; joints [-16.809, -38.616, 102.911, 144.694, 50.662, -28.556, -355]
  MoveL 4443 to (17.76, 73.23, -209.5) mm, rotated rx 42.04 ry 15.1 rz -114.75 deg; joints [-16.827, -38.53, 102.834, 144.677, 50.674, -28.555, -355]
  MoveL 4444 to (20.07, 73.52, -211.23) mm, rotated rx 42.04 ry 15.1 rz -114.75 deg; joints [-16.888, -38.371, 102.72, 144.626, 50.726, -28.561, -355]
  MoveL 4445 to (22.42, 73.02, -213.65) mm, rotated rx 42.04 ry 15.1 rz -114.75 deg; joints [-16.981, -38.228, 102.662, 144.555, 50.818, -28.581, -355]
  MoveL 4446 to (24.17, 71.99, -216.08) mm, rotated rx 42.04 ry 15.1 rz -114.75 deg; joints [-17.078, -38.138, 102.663, 144.483, 50.918, -28.607, -355]
  MoveL 4447 to (24.6, 71.37, -217.03) mm, rotated rx 42.04 ry 15.1 rz -114.75 deg; joints [-17.119, -38.124, 102.689, 144.454, 50.96, -28.618, -355]
  MoveL 4448 to (24.72, 70.69, -217.81) mm, rotated rx 42.04 ry 15.1 rz -114.75 deg; joints [-17.153, -38.132, 102.731, 144.429, 50.996, -28.628, -355]
  MoveL 4449 to (24.66, 70.32, -218.13) mm, rotated rx 42.04 ry 15.1 rz -114.75 deg; joints [-17.168, -38.144, 102.759, 144.418, 51.012, -28.632, -355]
  MoveL 4450 to (24.53, 69.94, -218.41) mm, rotated rx 42.04 ry 15.1 rz -114.75 deg; joints [-17.182, -38.162, 102.79, 144.408, 51.027, -28.637, -355]
  MoveL 4451 to (24.05, 69.12, -218.84) mm, rotated rx 42.04 ry 15.1 rz -114.75 deg; joints [-17.205, -38.212, 102.865, 144.392, 51.053, -28.645, -355]
  MoveL 4452 to (23.26, 68.24, -219.1) mm, rotated rx 42.04 ry 15.1 rz -114.75 deg; joints [-17.223, -38.285, 102.957, 144.38, 51.073, -28.651, -355]
  MoveL 4453 to (22.17, 67.28, -219.19) mm, rotated rx 42.04 ry 15.1 rz -114.75 deg; joints [-17.235, -38.379, 103.065, 144.373, 51.088, -28.657, -355]
  MoveL 4454 to (21.76, 66.96, -219.19) mm, rotated rx 42.04 ry 15.1 rz -114.75 deg; joints [-17.238, -38.413, 103.104, 144.371, 51.092, -28.658, -355]
  MoveL 4455 to (21.39, 66.69, -219.16) mm, rotated rx 42.04 ry 15.1 rz -114.75 deg; joints [-17.239, -38.444, 103.137, 144.371, 51.094, -28.66, -355]
  MoveL 4456 to (21.03, 66.45, -219.12) mm, rotated rx 42.04 ry 15.1 rz -114.75 deg; joints [-17.24, -38.473, 103.167, 144.371, 51.095, -28.66, -355]
  MoveL 4457 to (20.67, 66.23, -219.06) mm, rotated rx 42.04 ry 15.1 rz -114.75 deg; joints [-17.24, -38.501, 103.197, 144.371, 51.096, -28.661, -355]
  MoveL 4458 to (20.3, 65.97, -219.02) mm, rotated rx 42.04 ry 15.1 rz -114.75 deg; joints [-17.241, -38.532, 103.229, 144.371, 51.098, -28.662, -355]
  MoveL 4459 to (19.89, 65.66, -219) mm, rotated rx 42.04 ry 15.1 rz -114.75 deg; joints [-17.243, -38.566, 103.266, 144.37, 51.101, -28.663, -355]
  MoveL 4460 to (19.48, 65.34, -219) mm, rotated rx 42.04 ry 15.1 rz -114.75 deg; joints [-17.246, -38.6, 103.304, 144.368, 51.105, -28.665, -355]
  MoveL 4461 to (19.09, 65.03, -218.99) mm, rotated rx 42.04 ry 15.1 rz -114.75 deg; joints [-17.249, -38.633, 103.341, 144.367, 51.108, -28.666, -355]
  MoveL 4462 to (18.71, 64.75, -218.97) mm, rotated rx 42.04 ry 15.1 rz -114.75 deg; joints [-17.25, -38.664, 103.375, 144.366, 51.111, -28.668, -355]
  MoveL 4463 to (18.36, 64.5, -218.92) mm, rotated rx 42.04 ry 15.1 rz -114.75 deg; joints [-17.251, -38.693, 103.405, 144.367, 51.112, -28.669, -355]
  MoveL 4464 to (18.01, 64.27, -218.86) mm, rotated rx 42.04 ry 15.1 rz -114.75 deg; joints [-17.251, -38.722, 103.435, 144.367, 51.113, -28.67, -355]
  MoveL 4465 to (17.62, 64.01, -218.8) mm, rotated rx 42.04 ry 15.1 rz -114.75 deg; joints [-17.251, -38.753, 103.469, 144.368, 51.115, -28.671, -355]
  MoveL 4466 to (17.13, 63.65, -218.77) mm, rotated rx 42.04 ry 15.1 rz -114.75 deg; joints [-17.253, -38.794, 103.513, 144.367, 51.118, -28.672, -355]
  MoveL 4467 to (16.49, 63.18, -218.75) mm, rotated rx 42.04 ry 15.1 rz -114.75 deg; joints [-17.256, -38.847, 103.569, 144.364, 51.122, -28.674, -355]
  MoveL 4468 to (15.26, 62.2, -218.75) mm, rotated rx 42.04 ry 15.1 rz -114.75 deg; joints [-17.266, -38.95, 103.683, 144.359, 51.133, -28.678, -355]
  MoveL 4469 to (14.6, 61.7, -218.71) mm, rotated rx 42.04 ry 15.1 rz -114.75 deg; joints [-17.269, -39.006, 103.744, 144.357, 51.138, -28.68, -355]
  MoveL 4470 to (14.1, 61.32, -218.7) mm, rotated rx 42.04 ry 15.1 rz -114.75 deg; joints [-17.272, -39.047, 103.789, 144.355, 51.142, -28.681, -355]
  MoveL 4471 to (13.68, 61.05, -218.7) mm, rotated rx 42.04 ry 15.1 rz -114.75 deg; joints [-17.274, -39.08, 103.822, 144.352, 51.142, -28.68, -355]
  MoveL 4472 to (13.31, 60.86, -218.67) mm, rotated rx 42.04 ry 15.1 rz -114.75 deg; joints [-17.275, -39.108, 103.848, 144.35, 51.141, -28.678, -355]
  MoveL 4473 to (13.11, 60.81, -218.57) mm, rotated rx 42.04 ry 15.1 rz -114.75 deg; joints [-17.272, -39.123, 103.859, 144.353, 51.137, -28.677, -355]
  MoveL 4474 to (13.15, 60.87, -218.35) mm, rotated rx 42.04 ry 15.1 rz -114.75 deg; joints [-17.263, -39.121, 103.857, 144.363, 51.135, -28.681, -355]
  MoveL 4475 to (13.43, 61.05, -218) mm, rotated rx 42.04 ry 15.1 rz -114.75 deg; joints [-17.248, -39.101, 103.842, 144.383, 51.135, -28.691, -355]
  MoveL 4476 to (12.78, 61.49, -217.3) mm, rotated rx 42.04 ry 15.1 rz -114.75 deg; joints [-17.219, -39.131, 103.832, 144.399, 51.095, -28.675, -355]
  MoveL 4477 to (10.78, 61.37, -217.14) mm, rotated rx 42.04 ry 15.1 rz -114.75 deg; joints [-17.215, -39.255, 103.891, 144.372, 51.041, -28.627, -355]
  MoveL 4478 to (8.86, 61.3, -216.86) mm, rotated rx 42.04 ry 15.1 rz -114.75 deg; joints [-17.207, -39.374, 103.947, 144.353, 50.988, -28.584, -355]
  MoveL 4479 to (6.93, 61.19, -216.59) mm, rotated rx 42.04 ry 15.1 rz -114.75 deg; joints [-17.198, -39.494, 104.004, 144.333, 50.935, -28.541, -355]
  MoveL 4480 to (5, 61.08, -216.32) mm, rotated rx 42.04 ry 15.1 rz -114.75 deg; joints [-17.191, -39.614, 104.062, 144.313, 50.883, -28.498, -355]
  MoveL 4481 to (2.97, 60.96, -216.1) mm, rotated rx 42.04 ry 15.1 rz -114.75 deg; joints [-17.185, -39.74, 104.121, 144.289, 50.827, -28.451, -355]
  MoveL 4482 to (0.85, 60.9, -215.96) mm, rotated rx 42.04 ry 15.1 rz -114.75 deg; joints [-17.181, -39.868, 104.176, 144.258, 50.767, -28.396, -355]
  MoveL 4483 to (-1.68, 60.93, -215.85) mm, rotated rx 42.04 ry 15.1 rz -114.75 deg; joints [-17.179, -40.018, 104.23, 144.215, 50.688, -28.325, -355]
  MoveL 4484 to (-4.15, 60.61, -215.78) mm, rotated rx 42.04 ry 15.1 rz -114.75 deg; joints [-17.18, -40.175, 104.313, 144.178, 50.629, -28.269, -355]
  MoveL 4485 to (-6.25, 60.33, -215.66) mm, rotated rx 42.04 ry 15.1 rz -114.75 deg; joints [-17.179, -40.309, 104.384, 144.148, 50.578, -28.222, -355]
  MoveL 4486 to (-8.13, 60.14, -215.48) mm, rotated rx 42.04 ry 15.1 rz -114.75 deg; joints [-17.176, -40.428, 104.445, 144.125, 50.529, -28.179, -355]
  MoveL 4487 to (-10.16, 59.96, -215.36) mm, rotated rx 42.04 ry 15.1 rz -114.75 deg; joints [-17.174, -40.554, 104.505, 144.095, 50.475, -28.13, -355]
  MoveL 4488 to (-12.24, 59.79, -215.22) mm, rotated rx 42.04 ry 15.1 rz -114.75 deg; joints [-17.171, -40.683, 104.566, 144.065, 50.419, -28.079, -355]
  MoveL 4489 to (-14.4, 59.62, -215.16) mm, rotated rx 42.04 ry 15.1 rz -114.75 deg; joints [-17.172, -40.817, 104.627, 144.029, 50.361, -28.023, -355]
  MoveL 4490 to (-16.53, 59.44, -214.93) mm, rotated rx 42.04 ry 15.1 rz -114.75 deg; joints [-17.166, -40.95, 104.691, 144.002, 50.303, -27.973, -355]
  MoveL 4491 to (-18.66, 59.26, -214.82) mm, rotated rx 42.04 ry 15.1 rz -114.75 deg; joints [-17.165, -41.082, 104.752, 143.969, 50.245, -27.919, -355]
  MoveL 4492 to (-20.78, 59.07, -214.6) mm, rotated rx 42.04 ry 15.1 rz -114.75 deg; joints [-17.159, -41.216, 104.816, 143.942, 50.188, -27.869, -355]
  MoveL 4493 to (-22.91, 58.88, -214.49) mm, rotated rx 42.04 ry 15.1 rz -114.75 deg; joints [-17.158, -41.348, 104.877, 143.908, 50.13, -27.815, -355]
  MoveL 4494 to (-25.04, 58.68, -214.27) mm, rotated rx 42.04 ry 15.1 rz -114.75 deg; joints [-17.153, -41.481, 104.942, 143.88, 50.073, -27.764, -355]
  MoveL 4495 to (-27.16, 58.49, -214.16) mm, rotated rx 42.04 ry 15.1 rz -114.75 deg; joints [-17.152, -41.613, 105.002, 143.846, 50.015, -27.71, -355]
  MoveL 4496 to (-29.29, 58.3, -214.05) mm, rotated rx 42.04 ry 15.1 rz -114.75 deg; joints [-17.151, -41.745, 105.062, 143.812, 49.957, -27.655, -355]
  MoveL 4497 to (-31.19, 58.06, -213.82) mm, rotated rx 42.04 ry 15.1 rz -114.75 deg; joints [-17.145, -41.866, 105.124, 143.789, 49.907, -27.612, -355]
  MoveL 4498 to (-33, 57.8, -213.52) mm, rotated rx 42.04 ry 15.1 rz -114.75 deg; joints [-17.137, -41.984, 105.188, 143.772, 49.862, -27.574, -355]
  MoveL 4499 to (-34.78, 57.5, -213.13) mm, rotated rx 42.04 ry 15.1 rz -114.75 deg; joints [-17.126, -42.101, 105.256, 143.761, 49.819, -27.541, -355]
  MoveL 4500 to (-33.37, 57.33, -212.2) mm, rotated rx 42.04 ry 15.1 rz -114.75 deg; joints [-17.092, -42.031, 105.262, 143.84, 49.871, -27.616, -355]
  MoveL 4501 to (-33.73, 57.31, -212.15) mm, rotated rx 42.04 ry 15.1 rz -114.75 deg; joints [-17.09, -42.054, 105.272, 143.836, 49.861, -27.607, -355]
  MoveL 4502 to (-34.1, 57.32, -212.09) mm, rotated rx 42.04 ry 15.1 rz -114.75 deg; joints [-17.088, -42.076, 105.279, 143.831, 49.848, -27.597, -355]
  MoveL 4503 to (-34.51, 57.41, -212.06) mm, rotated rx 42.04 ry 15.1 rz -114.75 deg; joints [-17.086, -42.097, 105.28, 143.823, 49.831, -27.582, -355]
  MoveL 4504 to (-34.93, 57.56, -212.03) mm, rotated rx 42.04 ry 15.1 rz -114.75 deg; joints [-17.084, -42.117, 105.275, 143.812, 49.811, -27.564, -355]
  MoveL 4505 to (-35.39, 57.78, -212.03) mm, rotated rx 42.04 ry 15.1 rz -114.75 deg; joints [-17.082, -42.137, 105.264, 143.8, 49.786, -27.541, -355]
  MoveL 4506 to (-35.84, 58.02, -212.02) mm, rotated rx 42.04 ry 15.1 rz -114.75 deg; joints [-17.08, -42.155, 105.252, 143.786, 49.76, -27.518, -355]
  MoveL 4507 to (-36.76, 58.54, -212.02) mm, rotated rx 42.04 ry 15.1 rz -114.75 deg; joints [-17.077, -42.192, 105.224, 143.758, 49.706, -27.469, -355]
  MoveL 4508 to (-37.19, 58.76, -212) mm, rotated rx 42.04 ry 15.1 rz -114.75 deg; joints [-17.074, -42.21, 105.212, 143.746, 49.682, -27.447, -355]
  MoveL 4509 to (-37.62, 58.96, -211.95) mm, rotated rx 42.04 ry 15.1 rz -114.75 deg; joints [-17.071, -42.229, 105.204, 143.736, 49.659, -27.428, -355]
  MoveL 4510 to (-38.1, 59.17, -211.88) mm, rotated rx 42.04 ry 15.1 rz -114.75 deg; joints [-17.067, -42.251, 105.196, 143.727, 49.634, -27.407, -355]
  MoveL 4511 to (-38.62, 59.42, -211.81) mm, rotated rx 42.04 ry 15.1 rz -114.75 deg; joints [-17.063, -42.274, 105.185, 143.715, 49.605, -27.383, -355]
  MoveL 4512 to (-39.13, 59.68, -211.78) mm, rotated rx 42.04 ry 15.1 rz -114.75 deg; joints [-17.059, -42.295, 105.172, 143.701, 49.577, -27.357, -355]
  MoveL 4513 to (-39.61, 59.94, -211.77) mm, rotated rx 42.04 ry 15.1 rz -114.75 deg; joints [-17.057, -42.315, 105.158, 143.687, 49.55, -27.333, -355]
  MoveL 4514 to (-40.07, 60.2, -211.76) mm, rotated rx 42.04 ry 15.1 rz -114.75 deg; joints [-17.055, -42.333, 105.144, 143.673, 49.522, -27.308, -355]
  MoveL 4515 to (-40.99, 60.71, -211.76) mm, rotated rx 42.04 ry 15.1 rz -114.75 deg; joints [-17.051, -42.37, 105.115, 143.644, 49.469, -27.259, -355]
  MoveL 4516 to (-41.9, 61.19, -211.74) mm, rotated rx 42.04 ry 15.1 rz -114.75 deg; joints [-17.047, -42.408, 105.091, 143.618, 49.418, -27.213, -355]
  MoveL 4517 to (-44.19, 62.47, -211.74) mm, rotated rx 42.04 ry 15.1 rz -114.75 deg; joints [-17.038, -42.498, 105.019, 143.546, 49.285, -27.09, -355]
  MoveL 4518 to (-45.41, 63.23, -211.83) mm, rotated rx 42.04 ry 15.1 rz -114.75 deg; joints [-17.036, -42.543, 104.972, 143.502, 49.21, -27.019, -355]
  MoveL 4519 to (-46.33, 63.98, -212.09) mm, rotated rx 42.04 ry 15.1 rz -114.75 deg; joints [-17.04, -42.569, 104.917, 143.455, 49.146, -26.953, -355]
  MoveL 4520 to (-46.93, 64.7, -212.53) mm, rotated rx 42.04 ry 15.1 rz -114.75 deg; joints [-17.051, -42.576, 104.855, 143.407, 49.094, -26.893, -355]
  MoveL 4521 to (-47.11, 65.05, -212.81) mm, rotated rx 42.04 ry 15.1 rz -114.75 deg; joints [-17.059, -42.573, 104.821, 143.381, 49.072, -26.866, -355]
  MoveL 4522 to (-47.22, 65.4, -213.14) mm, rotated rx 42.04 ry 15.1 rz -114.75 deg; joints [-17.068, -42.564, 104.786, 143.356, 49.053, -26.84, -355]
  MoveL 4523 to (-47.19, 66.08, -213.93) mm, rotated rx 42.04 ry 15.1 rz -114.75 deg; joints [-17.092, -42.533, 104.709, 143.303, 49.023, -26.792, -355]
  MoveL 4524 to (-46.85, 66.74, -214.9) mm, rotated rx 42.04 ry 15.1 rz -114.75 deg; joints [-17.123, -42.483, 104.625, 143.249, 49.004, -26.75, -355]
  MoveL 4525 to (-45.24, 68, -217.35) mm, rotated rx 42.04 ry 15.1 rz -114.75 deg; joints [-17.203, -42.326, 104.435, 143.134, 49, -26.684, -355]
  MoveL 4526 to (-42.96, 68.83, -219.81) mm, rotated rx 42.04 ry 15.1 rz -114.75 deg; joints [-17.287, -42.145, 104.271, 143.042, 49.037, -26.656, -355]
  MoveL 4527 to (-40.6, 68.88, -221.56) mm, rotated rx 42.04 ry 15.1 rz -114.75 deg; joints [-17.351, -41.991, 104.187, 143.001, 49.111, -26.68, -355]
  MoveL 4528 to (-39.39, 68.61, -222.18) mm, rotated rx 42.04 ry 15.1 rz -114.75 deg; joints [-17.375, -41.925, 104.176, 143.001, 49.162, -26.712, -355]
  MoveL 4529 to (-38.16, 68.16, -222.61) mm, rotated rx 42.04 ry 15.1 rz -114.75 deg; joints [-17.394, -41.865, 104.185, 143.013, 49.222, -26.757, -355]
  MoveL 4530 to (-35.64, 66.66, -222.97) mm, rotated rx 42.04 ry 15.1 rz -114.75 deg; joints [-17.419, -41.766, 104.263, 143.076, 49.371, -26.886, -355]
  MoveL 4531 to (-33.52, 65.1, -222.96) mm, rotated rx 42.04 ry 15.1 rz -114.75 deg; joints [-17.431, -41.694, 104.362, 143.148, 49.51, -27.014, -355]
  MoveL 4532 to (-33.1, 64.78, -222.95) mm, rotated rx 42.04 ry 15.1 rz -114.75 deg; joints [-17.433, -41.68, 104.382, 143.164, 49.538, -27.041, -355]
  MoveL 4533 to (-32.68, 64.44, -222.92) mm, rotated rx 42.04 ry 15.1 rz -114.75 deg; joints [-17.434, -41.667, 104.405, 143.18, 49.567, -27.068, -355]
  MoveL 4534 to (-32.28, 64.14, -222.91) mm, rotated rx 42.04 ry 15.1 rz -114.75 deg; joints [-17.436, -41.654, 104.424, 143.194, 49.594, -27.093, -355]
  MoveL 4535 to (-31.92, 63.89, -222.93) mm, rotated rx 42.04 ry 15.1 rz -114.75 deg; joints [-17.439, -41.641, 104.439, 143.205, 49.617, -27.113, -355]
  MoveL 4536 to (-31.52, 63.61, -222.96) mm, rotated rx 42.04 ry 15.1 rz -114.75 deg; joints [-17.442, -41.626, 104.456, 143.217, 49.643, -27.136, -355]
  MoveL 4537 to (-31.03, 63.3, -223.02) mm, rotated rx 42.04 ry 15.1 rz -114.75 deg; joints [-17.447, -41.607, 104.472, 143.23, 49.673, -27.162, -355]
  MoveL 4538 to (-30.53, 63, -223.1) mm, rotated rx 42.04 ry 15.1 rz -114.75 deg; joints [-17.452, -41.588, 104.487, 143.241, 49.702, -27.187, -355]
  MoveL 4539 to (-30.06, 62.69, -223.15) mm, rotated rx 42.04 ry 15.1 rz -114.75 deg; joints [-17.456, -41.57, 104.505, 143.254, 49.731, -27.212, -355]
  MoveL 4540 to (-29.62, 62.39, -223.18) mm, rotated rx 42.04 ry 15.1 rz -114.75 deg; joints [-17.459, -41.554, 104.522, 143.267, 49.759, -27.237, -355]
  MoveL 4541 to (-29.2, 62.09, -223.19) mm, rotated rx 42.04 ry 15.1 rz -114.75 deg; joints [-17.462, -41.539, 104.541, 143.281, 49.787, -27.262, -355]
  MoveL 4542 to (-28.78, 61.78, -223.19) mm, rotated rx 42.04 ry 15.1 rz -114.75 deg; joints [-17.464, -41.525, 104.56, 143.295, 49.814, -27.287, -355]
  MoveL 4543 to (-28.31, 61.46, -223.22) mm, rotated rx 42.04 ry 15.1 rz -114.75 deg; joints [-17.468, -41.507, 104.578, 143.309, 49.844, -27.313, -355]
  MoveL 4544 to (-27.84, 61.17, -223.27) mm, rotated rx 42.04 ry 15.1 rz -114.75 deg; joints [-17.472, -41.489, 104.594, 143.321, 49.872, -27.338, -355]
  MoveL 4545 to (-27.35, 60.89, -223.34) mm, rotated rx 42.04 ry 15.1 rz -114.75 deg; joints [-17.477, -41.469, 104.607, 143.332, 49.9, -27.362, -355]
  MoveL 4546 to (-26.89, 60.69, -223.4) mm, rotated rx 42.04 ry 15.1 rz -114.75 deg; joints [-17.48, -41.448, 104.615, 143.342, 49.924, -27.383, -355]
  MoveL 4547 to (-26.45, 60.54, -223.43) mm, rotated rx 42.04 ry 15.1 rz -114.75 deg; joints [-17.483, -41.427, 104.619, 143.352, 49.945, -27.401, -355]
  MoveL 4548 to (-26.06, 60.48, -223.44) mm, rotated rx 42.04 ry 15.1 rz -114.75 deg; joints [-17.483, -41.406, 104.617, 143.361, 49.96, -27.416, -355]
  MoveL 4549 to (-25.67, 60.44, -223.44) mm, rotated rx 42.04 ry 15.1 rz -114.75 deg; joints [-17.483, -41.384, 104.612, 143.369, 49.974, -27.429, -355]
  MoveL 4550 to (-26.93, 60.72, -224.32) mm, rotated rx 42.04 ry 15.1 rz -114.75 deg; joints [-17.515, -41.441, 104.595, 143.294, 49.922, -27.355, -355]
  MoveL 4551 to (-25.33, 60.76, -224.6) mm, rotated rx 42.04 ry 15.1 rz -114.75 deg; joints [-17.524, -41.344, 104.554, 143.312, 49.97, -27.395, -355]
  MoveL 4552 to (-23.52, 60.76, -224.79) mm, rotated rx 42.04 ry 15.1 rz -114.75 deg; joints [-17.53, -41.236, 104.514, 143.338, 50.026, -27.446, -355]
  MoveL 4553 to (-21.47, 60.71, -224.92) mm, rotated rx 42.04 ry 15.1 rz -114.75 deg; joints [-17.534, -41.117, 104.475, 143.374, 50.092, -27.507, -355]
  MoveL 4554 to (-19.22, 60.62, -225.01) mm, rotated rx 42.04 ry 15.1 rz -114.75 deg; joints [-17.537, -40.987, 104.436, 143.416, 50.166, -27.576, -355]
  MoveL 4555 to (-17.09, 60.56, -225.16) mm, rotated rx 42.04 ry 15.1 rz -114.75 deg; joints [-17.541, -40.862, 104.395, 143.452, 50.234, -27.639, -355]
  MoveL 4556 to (-14.95, 60.51, -225.37) mm, rotated rx 42.04 ry 15.1 rz -114.75 deg; joints [-17.548, -40.736, 104.352, 143.485, 50.303, -27.699, -355]
  MoveL 4557 to (-12.93, 60.44, -225.5) mm, rotated rx 42.04 ry 15.1 rz -114.75 deg; joints [-17.552, -40.618, 104.314, 143.519, 50.368, -27.759, -355]
  MoveL 4558 to (-11.08, 60.4, -225.76) mm, rotated rx 42.04 ry 15.1 rz -114.75 deg; joints [-17.561, -40.508, 104.273, 143.543, 50.426, -27.809, -355]
  MoveL 4559 to (-9.01, 60.34, -225.98) mm, rotated rx 42.04 ry 15.1 rz -114.75 deg; joints [-17.568, -40.387, 104.231, 143.573, 50.492, -27.867, -355]
  MoveL 4560 to (-6.93, 60.26, -226.12) mm, rotated rx 42.04 ry 15.1 rz -114.75 deg; joints [-17.573, -40.265, 104.192, 143.608, 50.559, -27.928, -355]
  MoveL 4561 to (-4.8, 60.17, -226.22) mm, rotated rx 42.04 ry 15.1 rz -114.75 deg; joints [-17.576, -40.141, 104.152, 143.645, 50.628, -27.991, -355]
  MoveL 4562 to (-2.68, 60.09, -226.45) mm, rotated rx 42.04 ry 15.1 rz -114.75 deg; joints [-17.584, -40.016, 104.109, 143.676, 50.696, -28.05, -355]
  MoveL 4563 to (-0.53, 59.98, -226.71) mm, rotated rx 42.04 ry 15.1 rz -114.75 deg; joints [-17.593, -39.891, 104.067, 143.705, 50.765, -28.11, -355]
  MoveL 4564 to (1.59, 59.88, -226.8) mm, rotated rx 42.04 ry 15.1 rz -114.75 deg; joints [-17.596, -39.768, 104.028, 143.742, 50.834, -28.172, -355]
  MoveL 4565 to (3.76, 59.78, -226.84) mm, rotated rx 42.04 ry 15.1 rz -114.75 deg; joints [-17.597, -39.642, 103.988, 143.783, 50.904, -28.238, -355]
  MoveL 4566 to (5.87, 59.68, -226.95) mm, rotated rx 42.04 ry 15.1 rz -114.75 deg; joints [-17.6, -39.519, 103.949, 143.818, 50.972, -28.299, -355]
  MoveL 4567 to (7.99, 59.57, -227.15) mm, rotated rx 42.04 ry 15.1 rz -114.75 deg; joints [-17.608, -39.396, 103.908, 143.849, 51.04, -28.359, -355]
  MoveL 4568 to (10.06, 59.44, -227.48) mm, rotated rx 42.04 ry 15.1 rz -114.75 deg; joints [-17.62, -39.274, 103.865, 143.873, 51.107, -28.413, -355]
  MoveL 4569 to (12.21, 59.29, -227.74) mm, rotated rx 42.04 ry 15.1 rz -114.75 deg; joints [-17.629, -39.149, 103.824, 143.902, 51.178, -28.473, -355]
  MoveL 4570 to (14.34, 59.15, -227.94) mm, rotated rx 42.04 ry 15.1 rz -114.75 deg; joints [-17.637, -39.025, 103.785, 143.933, 51.247, -28.533, -355]
  MoveL 4571 to (16.51, 58.99, -228.18) mm, rotated rx 42.04 ry 15.1 rz -114.75 deg; joints [-17.645, -38.899, 103.744, 143.962, 51.319, -28.594, -355]
  MoveL 4572 to (18.66, 58.86, -228.32) mm, rotated rx 42.04 ry 15.1 rz -114.75 deg; joints [-17.65, -38.774, 103.703, 143.996, 51.388, -28.655, -355]
  MoveL 4573 to (20.77, 58.76, -228.34) mm, rotated rx 42.04 ry 15.1 rz -114.75 deg; joints [-17.651, -38.651, 103.662, 144.034, 51.454, -28.717, -355]
  MoveL 4574 to (21.27, 58.36, -229.01) mm, rotated rx 42.04 ry 15.1 rz -114.75 deg; joints [-17.679, -38.628, 103.671, 144.016, 51.487, -28.729, -355]
  MoveL 4575 to (20.95, 58.29, -229.34) mm, rotated rx 42.04 ry 15.1 rz -114.75 deg; joints [-17.692, -38.646, 103.678, 143.995, 51.481, -28.714, -355]
  MoveL 4576 to (20.91, 58.28, -229.55) mm, rotated rx 42.04 ry 15.1 rz -114.75 deg; joints [-17.7, -38.648, 103.676, 143.984, 51.481, -28.708, -355]
  MoveL 4577 to (21.12, 58.32, -229.65) mm, rotated rx 42.04 ry 15.1 rz -114.75 deg; joints [-17.703, -38.633, 103.666, 143.982, 51.485, -28.71, -355]
  MoveL 4578 to (21.52, 58.46, -229.67) mm, rotated rx 42.04 ry 15.1 rz -114.75 deg; joints [-17.702, -38.605, 103.643, 143.986, 51.49, -28.715, -355]
  MoveC 4579 to (22.42, 58.93, -229.67) mm, rotated rx 42.04 ry 15.1 rz -114.75 deg; joints [-17.698, -38.536, 103.581, 143.994, 51.493, -28.721, -355] to (23.29, 59.45, -229.67) mm, rotated rx 42.04 ry 15.1 rz -114.75 deg; joints [-17.692, -38.469, 103.514, 144.001, 51.493, -28.724, -355]
  MoveL 4580 to (23.29, 59.45, -229.67) mm, rotated rx 42.04 ry 15.1 rz -114.75 deg; joints [-17.693, -38.468, 103.514, 144.001, 51.493, -28.724, -355]
  MoveL 4581 to (23.76, 59.72, -229.69) mm, rotated rx 42.04 ry 15.1 rz -114.75 deg; joints [-17.691, -38.432, 103.479, 144.004, 51.493, -28.726, -355]
  MoveL 4582 to (24.24, 59.98, -229.74) mm, rotated rx 42.04 ry 15.1 rz -114.75 deg; joints [-17.69, -38.395, 103.444, 144.005, 51.494, -28.727, -355]
  MoveL 4583 to (24.76, 60.24, -229.81) mm, rotated rx 42.04 ry 15.1 rz -114.75 deg; joints [-17.69, -38.356, 103.407, 144.007, 51.497, -28.729, -355]
  MoveL 4584 to (25.28, 60.53, -229.85) mm, rotated rx 42.04 ry 15.1 rz -114.75 deg; joints [-17.689, -38.316, 103.369, 144.009, 51.498, -28.731, -355]
  MoveL 4585 to (26.33, 61.14, -229.88) mm, rotated rx 42.04 ry 15.1 rz -114.75 deg; joints [-17.683, -38.234, 103.289, 144.016, 51.498, -28.735, -355]
  MoveL 4586 to (26.81, 61.41, -229.91) mm, rotated rx 42.04 ry 15.1 rz -114.75 deg; joints [-17.682, -38.197, 103.253, 144.019, 51.499, -28.737, -355]
  MoveL 4587 to (27.24, 61.61, -229.98) mm, rotated rx 42.04 ry 15.1 rz -114.75 deg; joints [-17.683, -38.164, 103.224, 144.019, 51.501, -28.739, -355]
  MoveL 4588 to (27.64, 61.79, -230.07) mm, rotated rx 42.04 ry 15.1 rz -114.75 deg; joints [-17.684, -38.134, 103.197, 144.019, 51.504, -28.74, -355]
  MoveL 4589 to (28.02, 61.98, -230.13) mm, rotated rx 42.04 ry 15.1 rz -114.75 deg; joints [-17.685, -38.105, 103.17, 144.019, 51.506, -28.742, -355]
  MoveL 4590 to (28.42, 62.19, -230.17) mm, rotated rx 42.04 ry 15.1 rz -114.75 deg; joints [-17.684, -38.075, 103.141, 144.02, 51.507, -28.743, -355]
  MoveL 4591 to (30.66, 63.55, -230.17) mm, rotated rx 42.04 ry 15.1 rz -114.75 deg; joints [-17.671, -37.9, 102.967, 144.037, 51.504, -28.749, -355]
  MoveL 4592 to (33.27, 64.82, -230.52) mm, rotated rx 42.04 ry 15.1 rz -114.75 deg; joints [-17.671, -37.702, 102.784, 144.043, 51.516, -28.76, -355]
  MoveL 4593 to (34.51, 65.18, -230.95) mm, rotated rx 42.04 ry 15.1 rz -114.75 deg; joints [-17.683, -37.614, 102.713, 144.037, 51.533, -28.768, -355]
  MoveL 4594 to (35.69, 65.34, -231.55) mm, rotated rx 42.04 ry 15.1 rz -114.75 deg; joints [-17.703, -37.534, 102.657, 144.025, 51.558, -28.778, -355]
  MoveL 4595 to (36.83, 65.31, -232.33) mm, rotated rx 42.04 ry 15.1 rz -114.75 deg; joints [-17.731, -37.461, 102.615, 144.006, 51.59, -28.789, -355]
  MoveL 4596 to (37.91, 65.1, -233.27) mm, rotated rx 42.04 ry 15.1 rz -114.75 deg; joints [-17.768, -37.395, 102.587, 143.981, 51.63, -28.802, -355]
  MoveL 4597 to (39.94, 64.1, -235.69) mm, rotated rx 42.04 ry 15.1 rz -114.75 deg; joints [-17.865, -37.284, 102.574, 143.912, 51.733, -28.833, -355]
  MoveL 4598 to (41.27, 62.73, -238.1) mm, rotated rx 42.04 ry 15.1 rz -114.75 deg; joints [-17.966, -37.226, 102.61, 143.837, 51.833, -28.86, -355]
  MoveL 4599 to (41.48, 62.06, -239.05) mm, rotated rx 42.04 ry 15.1 rz -114.75 deg; joints [-18.007, -37.226, 102.644, 143.805, 51.871, -28.868, -355]
  MoveL 4600 to (41.39, 61.38, -239.83) mm, rotated rx 42.04 ry 15.1 rz -114.75 deg; joints [-18.041, -37.246, 102.689, 143.776, 51.9, -28.872, -355]
  MoveL 4601 to (41.23, 61.05, -240.15) mm, rotated rx 42.04 ry 15.1 rz -114.75 deg; joints [-18.057, -37.262, 102.715, 143.763, 51.911, -28.873, -355]
  MoveL 4602 to (40.99, 60.72, -240.43) mm, rotated rx 42.04 ry 15.1 rz -114.75 deg; joints [-18.07, -37.284, 102.744, 143.75, 51.921, -28.873, -355]
  MoveL 4603 to (40.3, 60.05, -240.86) mm, rotated rx 42.04 ry 15.1 rz -114.75 deg; joints [-18.093, -37.342, 102.811, 143.728, 51.933, -28.87, -355]
  MoveL 4604 to (39.31, 59.39, -241.12) mm, rotated rx 42.04 ry 15.1 rz -114.75 deg; joints [-18.109, -37.419, 102.888, 143.709, 51.937, -28.863, -355]
  MoveL 4605 to (38.01, 58.73, -241.21) mm, rotated rx 42.04 ry 15.1 rz -114.75 deg; joints [-18.119, -37.516, 102.976, 143.693, 51.933, -28.852, -355]
